// TwinCAT 3 PLC project R2_SafetyPLC
// ProgramVersion: 3.1.4022.3
// libraries:
//   Tc2_EtherCAT, * (Beckhoff Automation GmbH)
//   Tc2_Standard, * (Beckhoff Automation GmbH)
//   Tc2_System, * (Beckhoff Automation GmbH)
//   Tc2_Utilities, * (Beckhoff Automation GmbH)
//   Tc3_Module, * (Beckhoff Automation GmbH)
//   VisuDialogs, * (System)
// project tree:
//   DUTs/FBs/Enums/ E_SAFETY_FBState.TcDUT, E_SAFETY_FBStateCS.TcDUT, E_SAFETY_FBStateMUTING.TcDUT, E_SAFETY_FBStateSetReset.TcDUT, E_SAFETY_FBStateTimer.TcDUT
//   DUTs/FBs/FBStatus/ ST_Empty.TcDUT, ST_SAFETY_AND.TcDUT, ST_SAFETY_CONNECTIONSHUTDOWN.TcDUT, ST_SAFETY_DECOUPLE.TcDUT, ST_SAFETY_EDM.TcDUT, ST_SAFETY_ESTOP.TcDUT, ST_SAFETY_FBStatus.TcDUT, ST_SAFETY_MON.TcDUT, ST_SAFETY_MUTING.TcDUT, ST_SAFETY_OPMODE.TcDUT, ST_SAFETY_OR.TcDUT, ST_SAFETY_RS.TcDUT, ST_SAFETY_SR.TcDUT, ST_SAFETY_TOF.TcDUT, ST_SAFETY_TON.TcDUT, ST_SAFETY_TWOHAND.TcDUT
//   DUTs/FBs/ ST_SAFETY_FBAND.TcDUT, ST_SAFETY_FBCONNECTIONSHUTDOWN.TcDUT, ST_SAFETY_FBDECOUPLE.TcDUT, ST_SAFETY_FBEDM.TcDUT, ST_SAFETY_FBESTOP.TcDUT, ST_SAFETY_FBMON.TcDUT, ST_SAFETY_FBMUTING.TcDUT, ST_SAFETY_FBOPMODE.TcDUT, ST_SAFETY_FBOR.TcDUT, ST_SAFETY_FBRS.TcDUT, ST_SAFETY_FBSR.TcDUT, ST_SAFETY_FBTOF.TcDUT, ST_SAFETY_FBTON.TcDUT, ST_SAFETY_FBTWOHAND.TcDUT
//   DUTs/FBs/Unions/ U_SAFETY_AND.TcDUT, U_SAFETY_CONNECTIONSHUTDOWN.TcDUT, U_SAFETY_DECOUPLE.TcDUT, U_SAFETY_EDM.TcDUT, U_SAFETY_ESTOP.TcDUT, U_SAFETY_MON.TcDUT, U_SAFETY_MUTING.TcDUT, U_SAFETY_OPMODE.TcDUT, U_SAFETY_OR.TcDUT, U_SAFETY_RS.TcDUT, U_SAFETY_SR.TcDUT, U_SAFETY_TOF.TcDUT, U_SAFETY_TON.TcDUT, U_SAFETY_TWOHAND.TcDUT
//   DUTs/HW/ E_AX580x_ERROR.TcDUT, ST_AX580x_DiagnosticData.TcDUT, ST_EL1904_DiagnosticData.TcDUT, ST_EL2904_DiagnosticData.TcDUT, ST_EL6900_DiagnosticData.TcDUT, ST_EL6900_StatusData.TcDUT, ST_ELxxxx_Data.TcDUT
//   DUTs/Others/ E_SAFETY_ConnectionDiag.TcDUT, E_SAFETY_ConnectionState.TcDUT, E_SAFETY_GroupState.TcDUT, E_SAFETY_ProjectState.TcDUT, ST_SAFETYGroupIO.TcDUT, ST_SAFETYStatusConnection.TcDUT, ST_SAFETYStatusGroup.TcDUT
//   / GlobalTextList.TcGTLO, SafetyTask.TcTTO, Visualization Manager.TcVMO (not stored)
//   POUs/FBs/ F_SAFETY_StatusFB_TO_AND.TcPOU, F_SAFETY_StatusFB_TO_CONNECTIONSHUTDOWN.TcPOU, F_SAFETY_StatusFB_TO_DECOUPLE.TcPOU, F_SAFETY_StatusFB_TO_EDM.TcPOU, F_SAFETY_StatusFB_TO_ESTOP.TcPOU, F_SAFETY_StatusFB_TO_MON.TcPOU, F_SAFETY_StatusFB_TO_MUTING.TcPOU, F_SAFETY_StatusFB_TO_OPMODE.TcPOU, F_SAFETY_StatusFB_TO_OR.TcPOU, F_SAFETY_StatusFB_TO_RS.TcPOU, F_SAFETY_StatusFB_TO_SR.TcPOU, F_SAFETY_StatusFB_TO_TOF.TcPOU, F_SAFETY_StatusFB_TO_TON.TcPOU, F_SAFETY_StatusFB_TO_TWOHAND.TcPOU
//   POUs/HW/ FB_AX580x_DiagnosticData.TcPOU, FB_EL1904_DiagnosticData.TcPOU, FB_EL2904_DiagnosticData.TcPOU, FB_EL6900_DiagnosticData.TcPOU, FB_EL6900_StatusData.TcPOU
//   POUs/ MAINSafety.TcPOU
//   POUs/Others/ FB_SAFETY_AutoGroupErrACK.TcPOU, F_SAFETY_DOUBLESWAPDWORD.TcPOU, F_SAFETY_DWORD_TO_STIRNGHEX.TcPOU, I_ErrorHandling.TcIO
//   Version/ F_GetVersionSafetyDiag.TcPOU, Global_Version.TcGVL
//   VISUs/FBs/ TL_ConnectionDiag.TcTLO, TL_ConnectionState.TcTLO, TL_FbState.TcTLO, TL_FbStateCS.TcTLO, TL_FbStateMUTING.TcTLO, TL_FbStateSetReset.TcTLO, TL_FbStateTimer.TcTLO, TL_GroupState.TcTLO, V_PH_AND.TcVIS, V_PH_CONNECTIONSHUTDOWN.TcVIS, V_PH_DECOUPLE.TcVIS, V_PH_EDM.TcVIS, V_PH_ESTOP.TcVIS, V_PH_MON.TcVIS, V_PH_MUTING.TcVIS, V_PH_OPMODE.TcVIS, V_PH_OR.TcVIS, V_PH_RS.TcVIS, V_PH_SR.TcVIS, V_PH_TOF.TcVIS, V_PH_TON.TcVIS, V_PH_TWOHAND.TcVIS
//   VISUs/HW/ V_PH_EL1904_DIAG.TcVIS, V_PH_EL2904_DIAG.TcVIS, V_PH_EL6900_DIAG.TcVIS
//   VISUs/ V_PH_CONNECTION.TcVIS, V_PH_GROUP.TcVIS
// (motion and I/O tree: see PLC project r1_templateplc)
// real-time tasks:
//   TASK PlcTask: cycle T#10ms, priority 20, ADS port 350
//   TASK SafetyTask: cycle T#10ms, priority 21, ADS port 351

CONFIGURATION R2_SafetyPLC
    RESOURCE PLC ON TwinCAT3
        TASK SafetyTask(INTERVAL := T#10ms, PRIORITY := 21);
        PROGRAM MAINSafety WITH SafetyTask : MAINSafety;
    END_RESOURCE
END_CONFIGURATION

// ---- DUTs/FBs/Enums/E_SAFETY_FBState.TcDUT
TYPE E_SAFETY_FBState :
(* Refers to the following function blocks: AND, OR, OPMODE, ESTOP, MON, DECOUPLE, TWO-HAND, EDM *)
(
	eSAFETY_FBState_UNDEFINED		:= 0,
	eSAFETY_FBState_RUN				:= 1,
	eSAFETY_FBState_STOP 			:= 2,
	eSAFETY_FBState_SAFE 			:= 3,
	eSAFETY_FBState_ERROR 			:= 4,
	eSAFETY_FBState_RESET 			:= 5,
	eSAFETY_FBState_START 			:= 6,
	eSAFETY_FBState_ERRORDELAY		:= 7,
	eSAFETY_FBState_DELAYOUT		:= 8,
	eSAFETY_FBState_FUNCTEST		:= 9,
	eSAFETY_FBState_1BUTTON			:= 11,
	eSAFETY_FBState_2BUTTON			:= 12,
	eSAFETY_FBState_RELEASE			:= 13,
	eSAFETY_FBState_MONOFF			:= 14,
	eSAFETY_FBState_MONON			:= 15
);
END_TYPE

// ---- DUTs/FBs/Enums/E_SAFETY_FBStateCS.TcDUT
TYPE E_SAFETY_FBStateCS :
(* Refers to the following function blocks: CONNECTION SHUTDOWN *)
(
	eSAFETY_FBStateCS_UNDEFINED			:= 0,
	eSAFETY_FBStateCS_RUN				:= 1,
	eSAFETY_FBStateCS_STOP 				:= 2,
	eSAFETY_FBStateCS_SAFE 				:= 3,
	eSAFETY_FBStateCS_ERROR 			:= 4,
	eSAFETY_FBStateCS_RESET				:= 5,
	eSAFETY_FBStateCS_ACTIVE			:= 10,
	eSAFETY_FBStateCS_DEACTIVE			:= 11
);
END_TYPE

// ---- DUTs/FBs/Enums/E_SAFETY_FBStateMUTING.TcDUT
TYPE E_SAFETY_FBStateMUTING :
(* Refers to the following function blocks: MUTING *)
(
	eSAFETY_FBStateMUTING_UNDEFINED		:= 0,
	eSAFETY_FBStateMUTING_RUN 			:= 1,
	eSAFETY_FBStateMUTING_STOP 			:= 2,
	eSAFETY_FBStateMUTING_SAFE 			:= 3,
	eSAFETY_FBStateMUTING_ERROR 		:= 4,
	eSAFETY_FBStateMUTING_RESET			:= 5,
	eSAFETY_FBStateMUTING_DELAYOUT		:= 8,
	eSAFETY_FBStateMUTING_MUTING1		:= 9,
	eSAFETY_FBStateMUTING_MUTING2		:= 10,
	eSAFETY_FBStateMUTING_MUTING3		:= 11,
	eSAFETY_FBStateMUTING_MUTING4		:= 12,
	eSAFETY_FBStateMUTING_MUTING5		:= 13,
	eSAFETY_FBStateMUTING_MUTING6		:= 14,
	eSAFETY_FBStateMUTING_MUTING7		:= 15,
	eSAFETY_FBStateMUTING_MUTING8		:= 16,
	eSAFETY_FBStateMUTING_MUTING9		:= 17
);
END_TYPE

// ---- DUTs/FBs/Enums/E_SAFETY_FBStateSetReset.TcDUT
TYPE E_SAFETY_FBStateSetReset :
(* Refers to the following function blocks: SR, RS *)
(
	eSAFETY_FBStateSetReset_UNDEFINED 	:= 0,
	eSAFETY_FBStateSetReset_STOP 		:= 2,
	eSAFETY_FBStateSetReset_SAFE 		:= 3,
	eSAFETY_FBStateSetReset_SET 		:= 9
);
END_TYPE

// ---- DUTs/FBs/Enums/E_SAFETY_FBStateTimer.TcDUT
TYPE E_SAFETY_FBStateTimer :
(* Refers to the following function blocks: TON, TOF *)
(
	eSAFETY_FBStateTimer_UNDEFINED 	:= 0,
	eSAFETY_FBStateTimer_RUN 		:= 1,
	eSAFETY_FBStateTimer_STOP 		:= 2,
	eSAFETY_FBStateTimer_SAFE 		:= 3,
	eSAFETY_FBStateTimer_DELAYOUT 	:= 8,
	eSAFETY_FBStateTimer_DELAYIN 	:= 9
);
END_TYPE

// ---- DUTs/FBs/FBStatus/ST_Empty.TcDUT
TYPE ST_Empty :
STRUCT
	{attribute 'hide'}
	BUnknown						: BYTE;
	BState							: BYTE;
(* wDiagnosis *)
	{attribute 'hide'}
	bDiagBIT0						: BIT; 		(* Empty *)
	{attribute 'hide'}
	bDiagBIT1						: BIT; 		(* Empty *)
	{attribute 'hide'}
	bDiagBIT2						: BIT; 		(* Empty *)
	{attribute 'hide'}
	bDiagBIT3						: BIT; 		(* Empty *)
	{attribute 'hide'}
	bDiagBIT4						: BIT; 		(* Empty *)
	{attribute 'hide'}
	bDiagBIT5						: BIT; 		(* Empty *)
	{attribute 'hide'}
	bDiagBIT6						: BIT; 		(* Empty *)
	{attribute 'hide'}
	bDiagBIT7						: BIT; 		(* Empty *)
	{attribute 'hide'}
	bDiagBIT8						: BIT; 		(* Empty *)
	{attribute 'hide'}
	bDiagBIT9						: BIT; 		(* Empty *)
	{attribute 'hide'}
	bDiagBIT10						: BIT; 		(* Empty *)
	{attribute 'hide'}
	bDiagBIT11						: BIT; 		(* Empty *)
	{attribute 'hide'}
	bDiagBIT12						: BIT; 		(* Empty *)
	{attribute 'hide'}
	bDiagBIT13						: BIT; 		(* Empty *)
	{attribute 'hide'}
	bDiagBIT14						: BIT; 		(* Empty *)
	{attribute 'hide'}
	bDiagBIT15						: BIT; 		(* Empty *)
(* wInputs *)
	{attribute 'hide'}
	bInputBIT0						: BIT; 		(* Empty *)
	{attribute 'hide'}
	bInputBIT1						: BIT; 		(* Empty *)
	{attribute 'hide'}
	bInputBIT2						: BIT; 		(* Empty *)
	{attribute 'hide'}
	bInputBIT3						: BIT; 		(* Empty *)
	{attribute 'hide'}
	bInputBIT4						: BIT; 		(* Empty *)
	{attribute 'hide'}
	bInputBIT5						: BIT; 		(* Empty *)
	{attribute 'hide'}
	bInputBIT6						: BIT; 		(* Empty *)
	{attribute 'hide'}
	bInputBIT7						: BIT; 		(* Empty *)
	{attribute 'hide'}
	bInputBIT8						: BIT; 		(* Empty *)
	{attribute 'hide'}
	bInputBIT9						: BIT; 		(* Empty *)
	{attribute 'hide'}
	bInputBIT10						: BIT; 		(* Empty *)
	{attribute 'hide'}
	bInputBIT11						: BIT; 		(* Empty *)
	{attribute 'hide'}
	bInputBIT12						: BIT; 		(* Empty *)
	{attribute 'hide'}
	bInputBIT13						: BIT; 		(* Empty *)
	{attribute 'hide'}
	bInputBIT14						: BIT; 		(* Empty *)
	{attribute 'hide'}
	bInputBIT15						: BIT; 		(* Empty *)
(* wOutputs *)
	{attribute 'hide'}
	bOutputBIT0						: BIT; 		(* Empty *)
	{attribute 'hide'}
	bOutputBIT1						: BIT; 		(* Empty *)
	{attribute 'hide'}
	bOutputBIT2						: BIT; 		(* Empty *)
	{attribute 'hide'}
	bOutputBIT3						: BIT; 		(* Empty *)
	{attribute 'hide'}
	bOutputBIT4						: BIT; 		(* Empty *)
	{attribute 'hide'}
	bOutputBIT5						: BIT; 		(* Empty *)
	{attribute 'hide'}
	bOutputBIT6						: BIT; 		(* Empty *)
	{attribute 'hide'}
	bOutputBIT7						: BIT; 		(* Empty *)
	{attribute 'hide'}
	bOutputBIT8						: BIT; 		(* Empty *)
	{attribute 'hide'}
	bOutputBIT9						: BIT; 		(* Empty *)
	{attribute 'hide'}
	bOutputBIT10					: BIT; 		(* Empty *)
	{attribute 'hide'}
	bOutputBIT11					: BIT; 		(* Empty *)
	{attribute 'hide'}
	bOutputBIT12					: BIT; 		(* Empty *)
	{attribute 'hide'}
	bOutputBIT13					: BIT; 		(* Empty *)
	{attribute 'hide'}
	bOutputBIT14					: BIT; 		(* Empty *)
	{attribute 'hide'}
	bOutputBIT15					: BIT; 		(* Empty *)
END_STRUCT
END_TYPE

// ---- DUTs/FBs/FBStatus/ST_SAFETY_AND.TcDUT
//UPDATE: Zamiana dwóch pierwszych bitów zmiennej wOutputs
TYPE ST_SAFETY_AND :
STRUCT
	{attribute 'hide'}
	BUnknown						: BYTE;
	BState							: BYTE;
(* wDiagnosis *)
	{attribute 'hide'}
	bDiagBIT0						: BIT; 		(* Empty *)
	{attribute 'hide'}
	bDiagBIT1						: BIT; 		(* Empty *)
	{attribute 'hide'}
	bDiagBIT2						: BIT; 		(* Empty *)
	{attribute 'hide'}
	bDiagBIT3						: BIT; 		(* Empty *)
	{attribute 'hide'}
	bDiagBIT4						: BIT; 		(* Empty *)
	{attribute 'hide'}
	bDiagBIT5						: BIT; 		(* Empty *)
	{attribute 'hide'}
	bDiagBIT6						: BIT; 		(* Empty *)
	{attribute 'hide'}
	bDiagBIT7						: BIT; 		(* Empty *)
	{attribute 'hide'}
	bDiagBIT8						: BIT; 		(* Empty *)
	{attribute 'hide'}
	bDiagBIT9						: BIT; 		(* Empty *)
	{attribute 'hide'}
	bDiagBIT10						: BIT; 		(* Empty *)
	{attribute 'hide'}
	bDiagBIT11						: BIT; 		(* Empty *)
	{attribute 'hide'}
	bDiagBIT12						: BIT; 		(* Empty *)
	{attribute 'hide'}
	bDiagBIT13						: BIT; 		(* Empty *)
	{attribute 'hide'}
	bDiagBIT14						: BIT; 		(* Empty *)
	{attribute 'hide'}
	bDiagBIT15						: BIT; 		(* Empty *)
(* wInputs *)
	{attribute 'hide'}
	bInputBIT0						: BIT; 		(* Empty *)
	{attribute 'hide'}
	bInputBIT1						: BIT; 		(* Empty *)
	{attribute 'hide'}
	bInputBIT2						: BIT; 		(* Empty *)
	{attribute 'hide'}
	bInputBIT3						: BIT; 		(* Empty *)
	{attribute 'hide'}
	bInputBIT4						: BIT; 		(* Empty *)
	{attribute 'hide'}
	bInputBIT5						: BIT; 		(* Empty *)
	{attribute 'hide'}
	bInputBIT6						: BIT; 		(* Empty *)
	{attribute 'hide'}
	bInputBIT7						: BIT; 		(* Empty *)
	bIn_ANDIn1						: BIT; 		(* .8 *)
	bIn_ANDIn2						: BIT; 		(* .9 *)
	bIn_ANDIn3						: BIT; 		(* .10 *)
	bIn_ANDIn4						: BIT; 		(* .11 *)
	bIn_ANDIn5						: BIT; 		(* .12 *)
	bIn_ANDIn6						: BIT; 		(* .13 *)
	bIn_ANDIn7						: BIT; 		(* .14 *)
	bIn_ANDIn8						: BIT; 		(* .15 *)
(* wOutputs *)
	{attribute 'hide'}
	bOut_ANDOut_OLD					: BIT; 		(* .0 UPDATE: Empty*)
	//{attribute 'hide'}
	bOut_ANDOut						: BIT; 		(* .1 UPDATE: AND_OUT*)
	{attribute 'hide'}
	bOutputBIT2						: BIT; 		(* Empty *)
	{attribute 'hide'}
	bOutputBIT3						: BIT; 		(* Empty *)
	{attribute 'hide'}
	bOutputBIT4						: BIT; 		(* Empty *)
	{attribute 'hide'}
	bOutputBIT5						: BIT; 		(* Empty *)
	{attribute 'hide'}
	bOutputBIT6						: BIT; 		(* Empty *)
	{attribute 'hide'}
	bOutputBIT7						: BIT; 		(* Empty *)
	{attribute 'hide'}
	bOutputBIT8						: BIT; 		(* Empty *)
	{attribute 'hide'}
	bOutputBIT9						: BIT; 		(* Empty *)
	{attribute 'hide'}
	bOutputBIT10					: BIT; 		(* Empty *)
	{attribute 'hide'}
	bOutputBIT11					: BIT; 		(* Empty *)
	{attribute 'hide'}
	bOutputBIT12					: BIT; 		(* Empty *)
	{attribute 'hide'}
	bOutputBIT13					: BIT; 		(* Empty *)
	{attribute 'hide'}
	bOutputBIT14					: BIT; 		(* Empty *)
	{attribute 'hide'}
	bOutputBIT15					: BIT; 		(* Empty *)
END_STRUCT
END_TYPE

// ---- DUTs/FBs/FBStatus/ST_SAFETY_CONNECTIONSHUTDOWN.TcDUT
TYPE ST_SAFETY_CONNECTIONSHUTDOWN :
STRUCT
	{attribute 'hide'}
	BUnknown						: BYTE;
	BState							: BYTE;
(* wDiagnosis *)
	
	bDiag_DiscErrorCS1_2			: BIT;  	(* Discrepancy error input group 1 *)
	{attribute 'hide'}
	bDiagBIT1						: BIT; 		(* Empty *)
	{attribute 'hide'}
	bDiagBIT2						: BIT; 		(* Empty *)
	{attribute 'hide'}
	bDiagBIT3						: BIT; 		(* Empty *)
	{attribute 'hide'}
	bDiagBIT4						: BIT; 		(* Empty *)
	{attribute 'hide'}
	bDiagBIT5						: BIT; 		(* Empty *)
	{attribute 'hide'}
	bDiagBIT6						: BIT; 		(* Empty *)
	{attribute 'hide'}
	bDiagBIT7						: BIT; 		(* Empty *)
	{attribute 'hide'}
	bDiagBIT8						: BIT; 		(* Empty *)
	{attribute 'hide'}
	bDiagBIT9						: BIT; 		(* Empty *)
	{attribute 'hide'}
	bDiagBIT10						: BIT; 		(* Empty *)
	{attribute 'hide'}
	bDiagBIT11						: BIT; 		(* Empty *)
	{attribute 'hide'}
	bDiagBIT12						: BIT; 		(* Empty *)
	{attribute 'hide'}
	bDiagBIT13						: BIT; 		(* Empty *)
	{attribute 'hide'}
	bDiagBIT14						: BIT; 		(* Empty *)
	{attribute 'hide'}
	bDiagBIT15						: BIT; 		(* Empty *)
(* wInputs *)
	{attribute 'hide'}
	bInputBIT0						: BIT; 		(* Empty *)
	{attribute 'hide'}
	bInputBIT1						: BIT; 		(* Empty *)
	{attribute 'hide'}
	bInputBIT2						: BIT; 		(* Empty *)
	{attribute 'hide'}
	bInputBIT3						: BIT; 		(* Empty *)
	{attribute 'hide'}
	bInputBIT4						: BIT; 		(* Empty *)
	{attribute 'hide'}
	bInputBIT5						: BIT; 		(* Empty *)
	{attribute 'hide'}
	bInputBIT6						: BIT; 		(* Empty *)
	{attribute 'hide'}
	bInputBIT7						: BIT; 		(* Empty *)
	bIn_Deactivate1					: BIT; 		(* .8 *)
	bIn_Deactivate2					: BIT; 		(* .9 *)
	{attribute 'hide'}
	bInputBIT10						: BIT; 		(* Empty *)
	{attribute 'hide'}
	bInputBIT11						: BIT; 		(* Empty *)
	{attribute 'hide'}
	bInputBIT12						: BIT; 		(* Empty *)
	{attribute 'hide'}
	bInputBIT13						: BIT; 		(* Empty *)
	{attribute 'hide'}
	bInputBIT14						: BIT; 		(* Empty *)
	{attribute 'hide'}
	bInputBIT15						: BIT; 		(* Empty *)
(* wOutputs *)
	bOut_Error						: BOOL; 	(* .0 *)
	bOut_Deactivated				: BOOL; 	(* .1 *)
	{attribute 'hide'}
	bOutputBIT2						: BIT; 		(* Empty *)
	{attribute 'hide'}
	bOutputBIT3						: BIT; 		(* Empty *)
	{attribute 'hide'}
	bOutputBIT4						: BIT; 		(* Empty *)
	{attribute 'hide'}
	bOutputBIT5						: BIT; 		(* Empty *)
	{attribute 'hide'}
	bOutputBIT6						: BIT; 		(* Empty *)
	{attribute 'hide'}
	bOutputBIT7						: BIT; 		(* Empty *)
	{attribute 'hide'}
	bOutputBIT8						: BIT; 		(* Empty *)
	{attribute 'hide'}
	bOutputBIT9						: BIT; 		(* Empty *)
	{attribute 'hide'}
	bOutputBIT10					: BIT; 		(* Empty *)
	{attribute 'hide'}
	bOutputBIT11					: BIT; 		(* Empty *)
	{attribute 'hide'}
	bOutputBIT12					: BIT; 		(* Empty *)
	{attribute 'hide'}
	bOutputBIT13					: BIT; 		(* Empty *)
	{attribute 'hide'}
	bOutputBIT14					: BIT; 		(* Empty *)
	{attribute 'hide'}
	bOutputBIT15					: BIT; 		(* Empty *)
END_STRUCT
END_TYPE

// ---- DUTs/FBs/FBStatus/ST_SAFETY_DECOUPLE.TcDUT
TYPE ST_SAFETY_DECOUPLE :
STRUCT
	{attribute 'hide'}
	BUnknown						: BYTE;
	BState							: BYTE;
(* wDiagnosis *)
	{attribute 'hide'}
	bDiagBIT0						: BIT; 		(* Empty *)
	{attribute 'hide'}
	bDiagBIT1						: BIT; 		(* Empty *)
	{attribute 'hide'}
	bDiagBIT2						: BIT; 		(* Empty *)
	{attribute 'hide'}
	bDiagBIT3						: BIT; 		(* Empty *)
	{attribute 'hide'}
	bDiagBIT4						: BIT; 		(* Empty *)
	{attribute 'hide'}
	bDiagBIT5						: BIT; 		(* Empty *)
	{attribute 'hide'}
	bDiagBIT6						: BIT; 		(* Empty *)
	{attribute 'hide'}
	bDiagBIT7						: BIT; 		(* Empty *)
	{attribute 'hide'}
	bDiagBIT8						: BIT; 		(* Empty *)
	{attribute 'hide'}
	bDiagBIT9						: BIT; 		(* Empty *)
	{attribute 'hide'}
	bDiagBIT10						: BIT; 		(* Empty *)
	{attribute 'hide'}
	bDiagBIT11						: BIT; 		(* Empty *)
	{attribute 'hide'}
	bDiagBIT12						: BIT; 		(* Empty *)
	{attribute 'hide'}
	bDiagBIT13						: BIT; 		(* Empty *)
	{attribute 'hide'}
	bDiagBIT14						: BIT; 		(* Empty *)
	{attribute 'hide'}
	bDiagBIT15						: BIT; 		(* Empty *)
(* wInputs *)
	{attribute 'hide'}
	bInputBIT0						: BIT; 		(* Empty *)
	{attribute 'hide'}
	bInputBIT1						: BIT; 		(* Empty *)
	{attribute 'hide'}
	bInputBIT2						: BIT; 		(* Empty *)
	{attribute 'hide'}
	bInputBIT3						: BIT; 		(* Empty *)
	{attribute 'hide'}
	bInputBIT4						: BIT; 		(* Empty *)
	{attribute 'hide'}
	bInputBIT5						: BIT; 		(* Empty *)
	{attribute 'hide'}
	bInputBIT6						: BIT; 		(* Empty *)
	{attribute 'hide'}
	bInputBIT7						: BIT; 		(* Empty *)
	bIn_DECOUPLEIn1					: BIT; 		(* .8 *)
	bIn_DECOUPLEIn2					: BIT; 		(* .9 *)
	bIn_DECOUPLEIn3					: BIT; 		(* .10 *)
	bIn_DECOUPLEIn4					: BIT; 		(* .11 *)
	bIn_DECOUPLEIn5					: BIT; 		(* .12 *)
	bIn_DECOUPLEIn6					: BIT; 		(* .13 *)
	bIn_DECOUPLEIn7					: BIT; 		(* .14 *)
	bIn_DECOUPLEIn8					: BIT; 		(* .15 *)
(* wOutputs *)
	{attribute 'hide'}
	bOutputBIT0						: BIT; 		(* Empty *)
	{attribute 'hide'}
	bOutputBIT1						: BIT; 		(* Empty *)
	{attribute 'hide'}
	bOutputBIT2						: BIT; 		(* Empty *)
	{attribute 'hide'}
	bOutputBIT3						: BIT; 		(* Empty *)
	{attribute 'hide'}
	bOutputBIT4						: BIT; 		(* Empty *)
	{attribute 'hide'}
	bOutputBIT5						: BIT; 		(* Empty *)
	{attribute 'hide'}
	bOutputBIT6						: BIT; 		(* Empty *)
	{attribute 'hide'}
	bOutputBIT7						: BIT; 		(* Empty *)
	bOut_DECOUPLEOut1				: BOOL; 	(* .8 *)
	bOut_DECOUPLEOut2				: BOOL; 	(* .9 *)
	bOut_DECOUPLEOut3				: BOOL; 	(* .10 *)
	bOut_DECOUPLEOut4				: BOOL; 	(* .11 *)
	bOut_DECOUPLEOut5				: BOOL; 	(* .12 *)
	bOut_DECOUPLEOut6				: BOOL; 	(* .13 *)
	bOut_DECOUPLEOut7				: BOOL; 	(* .14 *)
	bOut_DECOUPLEOut8				: BOOL; 	(* .15 *)
END_STRUCT
END_TYPE

// ---- DUTs/FBs/FBStatus/ST_SAFETY_EDM.TcDUT
TYPE ST_SAFETY_EDM :
STRUCT
	{attribute 'hide'}
	BUnknown						: BYTE;
	BState							: BYTE;
(* wDiagnosis *)
	bDiag_SwitchOffError			: BIT; 		(* Switch-OFF timer elapsed  *)
	bDiag_SwitchOnError				: BIT; 		(* Switch-ON timer elapsed  *)
	{attribute 'hide'}
	bDiagBIT2						: BIT; 		(* Empty *)
	{attribute 'hide'}
	bDiagBIT3						: BIT; 		(* Empty *)
	{attribute 'hide'}
	bDiagBIT4						: BIT; 		(* Empty *)
	{attribute 'hide'}
	bDiagBIT5						: BIT; 		(* Empty *)
	{attribute 'hide'}
	bDiagBIT6						: BIT; 		(* Empty *)
	{attribute 'hide'}
	bDiagBIT7						: BIT; 		(* Empty *)
	{attribute 'hide'}
	bDiagBIT8						: BIT; 		(* Empty *)
	{attribute 'hide'}
	bDiagBIT9						: BIT; 		(* Empty *)
	{attribute 'hide'}
	bDiagBIT10						: BIT; 		(* Empty *)
	{attribute 'hide'}
	bDiagBIT11						: BIT; 		(* Empty *)
	{attribute 'hide'}
	bDiagBIT12						: BIT; 		(* Empty *)
	{attribute 'hide'}
	bDiagBIT13						: BIT; 		(* Empty *)
	{attribute 'hide'}
	bDiagBIT14						: BIT; 		(* Empty *)
	{attribute 'hide'}
	bDiagBIT15						: BIT; 		(* Empty *)
(* wInputs *)
	{attribute 'hide'}
	bInputBIT0						: BIT; 		(* Empty *)
	{attribute 'hide'}
	bInputBIT1						: BIT; 		(* Empty *)
	{attribute 'hide'}
	bInputBIT2						: BIT; 		(* Empty *)
	{attribute 'hide'}
	bInputBIT3						: BIT; 		(* Empty *)
	{attribute 'hide'}
	bInputBIT4						: BIT; 		(* Empty *)
	{attribute 'hide'}
	bInputBIT5						: BIT; 		(* Empty *)
	{attribute 'hide'}
	bInputBIT6						: BIT; 		(* Empty *)
	{attribute 'hide'}
	bInputBIT7						: BIT; 		(* Empty *)
	bIn_MON1						: BIT; 		(* .8 *)
	bIn_MON2						: BIT; 		(* .9 *)
	{attribute 'hide'}
	bInputBIT10						: BIT; 		(* Empty *)
	{attribute 'hide'}
	bInputBIT11						: BIT; 		(* Empty *)
	{attribute 'hide'}
	bInputBIT12						: BIT; 		(* Empty *)
	{attribute 'hide'}
	bInputBIT13						: BIT; 		(* Empty *)
	{attribute 'hide'}
	bInputBIT14						: BIT; 		(* Empty *)
	{attribute 'hide'}
	bInputBIT15						: BIT; 		(* Empty *)
(* wOutputs *)
	bOut_Error						: BIT; 		(* .0 *)
	{attribute 'hide'}
	bOutputBIT1						: BIT; 		(* Empty *)
	{attribute 'hide'}
	bOutputBIT2						: BIT; 		(* Empty *)
	{attribute 'hide'}
	bOutputBIT3						: BIT; 		(* Empty *)
	{attribute 'hide'}
	bOutputBIT4						: BIT; 		(* Empty *)
	{attribute 'hide'}
	bOutputBIT5						: BIT; 		(* Empty *)
	{attribute 'hide'}
	bOutputBIT6						: BIT; 		(* Empty *)
	{attribute 'hide'}
	bOutputBIT7						: BIT; 		(* Empty *)
	{attribute 'hide'}
	bOutputBIT8						: BIT; 		(* Empty *)
	{attribute 'hide'}
	bOutputBIT9						: BIT; 		(* Empty *)
	{attribute 'hide'}
	bOutputBIT10					: BIT; 		(* Empty *)
	{attribute 'hide'}
	bOutputBIT11					: BIT; 		(* Empty *)
	{attribute 'hide'}
	bOutputBIT12					: BIT; 		(* Empty *)
	{attribute 'hide'}
	bOutputBIT13					: BIT; 		(* Empty *)
	{attribute 'hide'}
	bOutputBIT14					: BIT; 		(* Empty *)
	{attribute 'hide'}
	bOutputBIT15					: BIT; 		(* Empty *)
END_STRUCT
END_TYPE

// ---- DUTs/FBs/FBStatus/ST_SAFETY_ESTOP.TcDUT
TYPE ST_SAFETY_ESTOP :
STRUCT
	{attribute 'hide'}
	BUnknown						: BYTE;
	BState							: BYTE;
(* wDiagnosis *)
	bDiag_DiscError1_2				: BIT;		(* Bit 0: Discrepancy error input group 1 (EStopIn1/2) *)
	bDiag_DiscError3_4				: BIT;		(* Bit 1: Discrepancy error input group 2 (EStopIn3/4) *)
	bDiag_DiscError5_6				: BIT;		(* Bit 2: Discrepancy error input group 2 (EStopIn5/6) *)
	bDiag_DiscError7_8				: BIT;		(* Bit 3: Discrepancy error input group 2 (EStopIn7/8) *)
	bDiag_EDM1Error					: BIT;		(* Bit 4: EDM monitoring error EDM1 Error *)
	bDiag_EDM2Error					: BIT;		(* Bit 5: EDM monitoring error EDM2 Error *)
	{attribute 'hide'}
	bDiagBIT6						: BIT; 		(* Empty *)
	{attribute 'hide'}
	bDiagBIT7						: BIT; 		(* Empty *)
	bDiag_DiscErrorSIADE1_2			: BIT;		(* Bit 8: Discrepancy error input group 1 with activated option "Safe Inputs after Disc Error"  (set in addition to bit 0) *)
	bDiag_DiscErrorSIADE3_4			: BIT;		(* Bit 9: Discrepancy error input group 2 with activated option "Safe Inputs after Disc Error"  (set in addition to bit 1) *)
	bDiag_DiscErrorSIADE5_6			: BIT;		(* Bit 10: Discrepancy error input group 3 with activated option "Safe Inputs after Disc Error"  (set in addition to bit 2) *)
	bDiag_DiscErrorSIADE7_8			: BIT;		(* Bit 11: Discrepancy error input group 4 with activated option "Safe Inputs after Disc Error"  (set in addition to bit 3)*)
	{attribute 'hide'}
	bDiagBIT12						: BIT; 		(* Empty *)
	{attribute 'hide'}
	bDiagBIT13						: BIT; 		(* Empty *)
	{attribute 'hide'}
	bDiagBIT14						: BIT; 		(* Empty *)
	{attribute 'hide'}
	bDiagBIT15						: BIT; 		(* Empty *)
(* wInputs *)
	bIn_Restart						: BIT; 		(* .0 *)
	bIn_EDM1						: BIT; 		(* .1 *)
	bIn_EDM2						: BIT; 		(* .2 *)
	{attribute 'hide'}
	bInputBIT3						: BIT; 		(* Empty *)
	{attribute 'hide'}
	bInputBIT4						: BIT; 		(* Empty *)
	{attribute 'hide'}
	bInputBIT5						: BIT; 		(* Empty *)
	{attribute 'hide'}
	bInputBIT6						: BIT; 		(* Empty *)
	{attribute 'hide'}
	bInputBIT7						: BIT; 		(* Empty *)
	bIn_EStopIn1					: BIT; 		(* .8 *)
	bIn_EStopIn2					: BIT; 		(* .9 *)
	bIn_EStopIn3					: BIT; 		(* .10 *)
	bIn_EStopIn4					: BIT; 		(* .11 *)
	bIn_EStopIn5					: BIT; 		(* .12 *)
	bIn_EStopIn6					: BIT; 		(* .13 *)
	bIn_EStopIn7					: BIT; 		(* .14 *)
	bIn_EStopIn8					: BIT; 		(* .15 *)
(* wOutputs *)
	bOut_Error						: BIT; 		(* .0 *)
	bOut_EstopOut					: BIT; 		(* .1 *)
	bOut_EstopDelOut				: BIT; 		(* .2 *)
	{attribute 'hide'}
	bOutputBIT3						: BIT; 		(* Empty *)
	{attribute 'hide'}
	bOutputBIT4						: BIT; 		(* Empty *)
	{attribute 'hide'}
	bOutputBIT5						: BIT; 		(* Empty *)
	{attribute 'hide'}
	bOutputBIT6						: BIT; 		(* Empty *)
	{attribute 'hide'}
	bOutputBIT7						: BIT; 		(* Empty *)
	{attribute 'hide'}
	bOutputBIT8						: BIT; 		(* Empty *)
	{attribute 'hide'}
	bOutputBIT9						: BIT; 		(* Empty *)
	{attribute 'hide'}
	bOutputBIT10					: BIT; 		(* Empty *)
	{attribute 'hide'}
	bOutputBIT11					: BIT; 		(* Empty *)
	{attribute 'hide'}
	bOutputBIT12					: BIT; 		(* Empty *)
	{attribute 'hide'}
	bOutputBIT13					: BIT; 		(* Empty *)
	{attribute 'hide'}
	bOutputBIT14					: BIT; 		(* Empty *)
	{attribute 'hide'}
	bOutputBIT15					: BIT; 		(* Empty *)
END_STRUCT
END_TYPE

// ---- DUTs/FBs/FBStatus/ST_SAFETY_FBStatus.TcDUT
TYPE ST_SAFETY_FBStatus :
STRUCT
	BUnknown						: BYTE;
	BState							: BYTE;
	wDiagnosis						: WORD;
	wInputs							: WORD; (* 1B - Restart, EDM... 2B - Safe inputs *)
	wOutputs						: WORD; (* 1B - Error, EDM... 2B - Safe inputs  *)
END_STRUCT
END_TYPE

// ---- DUTs/FBs/FBStatus/ST_SAFETY_MON.TcDUT
TYPE ST_SAFETY_MON :
STRUCT
	{attribute 'hide'}
	BUnknown						: BYTE;
	BState							: BYTE;
(* wDiagnosis *)
	bDiag_DiscErrorMONIn1_2			: BIT; 		(* Discrepancy error input group 1 (MONIn1/2) *)
	bDiag_DiscErrorMONIn3_4			: BIT;		(* Discrepancy error input group 2 (MONIn3/4) *)
	bDiag_DiscErrorMONInSec			: BIT;		(* Discrepancy error in Secure input group (MONInSec)*) 
	{attribute 'hide'}
	bDiagBIT3						: BIT; 		(* Empty *)
	bDiag_EDM1Error					: BIT;		(* EDM monitoring error EDM1*)
	bDiag_EDM2Error					: BIT;		(* EDM monitoring error EDM2*) 
	{attribute 'hide'}
	bDiagBIT6						: BIT; 		(* Empty *)
	{attribute 'hide'}
	bDiagBIT7						: BIT; 		(* Empty *)
	{attribute 'hide'}
	bDiagBIT8						: BIT; 		(* Empty *)
	{attribute 'hide'}
	bDiagBIT9						: BIT; 		(* Empty *)
	{attribute 'hide'}
	bDiagBIT10						: BIT; 		(* Empty *)
	{attribute 'hide'}
	bDiagBIT11						: BIT; 		(* Empty *)
	{attribute 'hide'}
	bDiagBIT12						: BIT; 		(* Empty *)
	{attribute 'hide'}
	bDiagBIT13						: BIT; 		(* Empty *)
	{attribute 'hide'}
	bDiagBIT14						: BIT; 		(* Empty *)
	{attribute 'hide'}
	bDiagBIT15						: BIT; 		(* Empty *)
(* wInputs *)
	bIn_Restart						: BIT; 		(* .0 *)
	bIn_EDM1						: BIT; 		(* .1 *)
	bIn_EDM2						: BIT; 		(* .2 *)
	bIn_MONSec1						: BIT; 		(* .3 *)
	bIn_MONSec2						: BIT; 		(* .4 *)
	{attribute 'hide'}
	bInputBIT5						: BIT; 		(* Empty *)
	{attribute 'hide'}
	bInputBIT6						: BIT; 		(* Empty *)
	{attribute 'hide'}
	bInputBIT7						: BIT; 		(* Empty *)
	bIn_MONIn1						: BIT; 		(* .8 *)
	bIn_MONIn2						: BIT; 		(* .9 *)
	bIn_MONIn3						: BIT; 		(* .10 *)
	bIn_MONIn4						: BIT; 		(* .11 *)
	{attribute 'hide'}
	bInputBIT12						: BIT; 		(* Empty *)
	{attribute 'hide'}
	bInputBIT13						: BIT; 		(* Empty *)
	{attribute 'hide'}
	bInputBIT14						: BIT; 		(* Empty *)
	{attribute 'hide'}
	bInputBIT15						: BIT; 		(* Empty *)
(* wOutputs *)
	bOut_Error						: BIT; 		(* .0 *)
	bOut_MONOut						: BIT; 		(* .1 *)
	bOut_MONDelOut					: BIT; 		(* .2 *)
	{attribute 'hide'}
	bOutputBIT3						: BIT; 		(* Empty *)
	{attribute 'hide'}
	bOutputBIT4						: BIT; 		(* Empty *)
	{attribute 'hide'}
	bOutputBIT5						: BIT; 		(* Empty *)
	{attribute 'hide'}
	bOutputBIT6						: BIT; 		(* Empty *)
	{attribute 'hide'}
	bOutputBIT7						: BIT; 		(* Empty *)
	{attribute 'hide'}
	bOutputBIT8						: BIT; 		(* Empty *)
	{attribute 'hide'}
	bOutputBIT9						: BIT; 		(* Empty *)
	{attribute 'hide'}
	bOutputBIT10					: BIT; 		(* Empty *)
	{attribute 'hide'}
	bOutputBIT11					: BIT; 		(* Empty *)
	{attribute 'hide'}
	bOutputBIT12					: BIT; 		(* Empty *)
	{attribute 'hide'}
	bOutputBIT13					: BIT; 		(* Empty *)
	{attribute 'hide'}
	bOutputBIT14					: BIT; 		(* Empty *)
	{attribute 'hide'}
	bOutputBIT15					: BIT; 		(* Empty *)
END_STRUCT
END_TYPE

// ---- DUTs/FBs/FBStatus/ST_SAFETY_MUTING.TcDUT
TYPE ST_SAFETY_MUTING :
STRUCT
	{attribute 'hide'}
	BUnknown						: BYTE;
	BState							: BYTE;
(* wDiagnosis *)
	bDiag_DiscErrorMUTINGIn1_2		: BIT;		(*	Discrepancy error in muting input group 1 *)
	bDiag_DiscErrorMUTINGInOSSD		: BIT;		(*	Discrepancy error in the OSSD input group *)
	bDiag_DiscErrorMUTINGIn3_4		: BIT;		(*	Discrepancy error in muting input group 2 *)
	{attribute 'hide'}
	bDiagBIT3						: BIT; 		(* Empty *)
	bDiag_EDM1Error					: BIT;		(*	Bit 4: EDM monitoring error EDM1 Error *)
	bDiag_EDM2Error					: BIT;		(*	Bit 5: EDM monitoring error EDM2 Error *)
	bDiag_MutingSeqViolated			: BIT;		(*	Bit 6: Muting sequence was violated *)
	bDiag_MutingTimeExceeded		: BIT;		(*	Bit 7: Maximum muting time was exceeded *)
	{attribute 'hide'}
	bDiagBIT8						: BIT; 		(* Empty *)
	{attribute 'hide'}
	bDiagBIT9						: BIT; 		(* Empty *)
	{attribute 'hide'}
	bDiagBIT10						: BIT; 		(* Empty *)
	{attribute 'hide'}
	bDiagBIT11						: BIT; 		(* Empty *)
	{attribute 'hide'}
	bDiagBIT12						: BIT; 		(* Empty *)
	{attribute 'hide'}
	bDiagBIT13						: BIT; 		(* Empty *)
	{attribute 'hide'}
	bDiagBIT14						: BIT; 		(* Empty *)
	{attribute 'hide'}
	bDiagBIT15						: BIT; 		(* Empty *)
(* wInputs *)
	bIn_Enable						: BIT; 		(* .0 *)
	bIn_EDM1						: BIT; 		(* .1 *)
	bIn_EDM2						: BIT; 		(* .2 *)
	{attribute 'hide'}
	bInputBIT3						: BIT; 		(* Empty *)
	{attribute 'hide'}
	bInputBIT4						: BIT; 		(* Empty *)
	{attribute 'hide'}
	bInputBIT5						: BIT; 		(* Empty *)
	{attribute 'hide'}
	bInputBIT6						: BIT; 		(* Empty *)
	{attribute 'hide'}
	bInputBIT7						: BIT; 		(* Empty *)
	bIn_MUTINGIn1					: BIT; 		(* .8 *)
	bIn_MUTINGIn2					: BIT; 		(* .9 *)
	bIn_MUTINGIn3					: BIT; 		(* .10 *)
	bIn_MUTINGIn4					: BIT; 		(* .11 *)
	bIn_OSSDIn1						: BIT; 		(* .12 *)
	bIn_OSSDIn2						: BIT; 		(* .13 *)
	{attribute 'hide'}
	bInputBIT14						: BIT; 		(* Empty *)
	{attribute 'hide'}
	bInputBIT15						: BIT; 		(* Empty *)
(* wOutputs *)
	bOut_Error						: BIT; 		(* .0 *)
	bOut_MUTINGActive				: BIT; 		(* .1 *)
	bOut_MUTINGOut					: BIT; 		(* .2 *)
	bOut_MUTINGDelOut				: BIT; 		(* .3 *)
	{attribute 'hide'}
	bOutputBIT4						: BIT; 		(* Empty *)
	{attribute 'hide'}
	bOutputBIT5						: BIT; 		(* Empty *)
	{attribute 'hide'}
	bOutputBIT6						: BIT; 		(* Empty *)
	{attribute 'hide'}
	bOutputBIT7						: BIT; 		(* Empty *)
	{attribute 'hide'}
	bOutputBIT8						: BIT; 		(* Empty *)
	{attribute 'hide'}
	bOutputBIT9						: BIT; 		(* Empty *)
	{attribute 'hide'}
	bOutputBIT10					: BIT; 		(* Empty *)
	{attribute 'hide'}
	bOutputBIT11					: BIT; 		(* Empty *)
	{attribute 'hide'}
	bOutputBIT12					: BIT; 		(* Empty *)
	{attribute 'hide'}
	bOutputBIT13					: BIT; 		(* Empty *)
	{attribute 'hide'}
	bOutputBIT14					: BIT; 		(* Empty *)
	{attribute 'hide'}
	bOutputBIT15					: BIT; 		(* Empty *)
END_STRUCT
END_TYPE

// ---- DUTs/FBs/FBStatus/ST_SAFETY_OPMODE.TcDUT
TYPE ST_SAFETY_OPMODE :
STRUCT
	{attribute 'hide'}
	BUnknown						: BYTE;
	BState							: BYTE;
(* wDiagnosis *)
	bDiag_DiscError					: BIT; 		(* Discrepancy monitoring error *)
	{attribute 'hide'}
	bDiagBIT1						: BIT; 		(* Empty *)
	{attribute 'hide'}
	bDiagBIT2						: BIT; 		(* Empty *)
	{attribute 'hide'}
	bDiagBIT3						: BIT; 		(* Empty *)
	{attribute 'hide'}
	bDiagBIT4						: BIT; 		(* Empty *)
	{attribute 'hide'}
	bDiagBIT5						: BIT; 		(* Empty *)
	{attribute 'hide'}
	bDiagBIT6						: BIT; 		(* Empty *)
	{attribute 'hide'}
	bDiagBIT7						: BIT; 		(* Empty *)
	{attribute 'hide'}
	bDiagBIT8						: BIT; 		(* Empty *)
	{attribute 'hide'}
	bDiagBIT9						: BIT; 		(* Empty *)
	{attribute 'hide'}
	bDiagBIT10						: BIT; 		(* Empty *)
	{attribute 'hide'}
	bDiagBIT11						: BIT; 		(* Empty *)
	{attribute 'hide'}
	bDiagBIT12						: BIT; 		(* Empty *)
	{attribute 'hide'}
	bDiagBIT13						: BIT; 		(* Empty *)
	{attribute 'hide'}
	bDiagBIT14						: BIT; 		(* Empty *)
	{attribute 'hide'}
	bDiagBIT15						: BIT; 		(* Empty *)
(* wInputs *)
	bIn_Restart						: BIT; 		(* .0 *)
	{attribute 'hide'}
	bInputBIT1						: BIT; 		(* Empty *)
	{attribute 'hide'}
	bInputBIT2						: BIT; 		(* Empty *)
	{attribute 'hide'}
	bInputBIT3						: BIT; 		(* Empty *)
	{attribute 'hide'}
	bInputBIT4						: BIT; 		(* Empty *)
	{attribute 'hide'}
	bInputBIT5						: BIT; 		(* Empty *)
	{attribute 'hide'}
	bInputBIT6						: BIT; 		(* Empty *)
	{attribute 'hide'}
	bInputBIT7						: BIT; 		(* Empty *)
	bIn_OPMODEIn1					: BIT; 		(* .8 *)
	bIn_OPMODEIn2					: BIT; 		(* .9 *)
	bIn_OPMODEIn3					: BIT; 		(* .10 *)
	bIn_OPMODEIn4					: BIT; 		(* .11 *)
	bIn_OPMODEIn5					: BIT; 		(* .12 *)
	bIn_OPMODEIn6					: BIT; 		(* .13 *)
	bIn_OPMODEIn7					: BIT; 		(* .14 *)
	bIn_OPMODEIn8					: BIT; 		(* .15 *)
(* wOutputs *)
	bOut_Error						: BIT; 		(* .0 *)
	{attribute 'hide'}
	bOutputBIT1						: BIT; 		(* Empty *)
	{attribute 'hide'}
	bOutputBIT2						: BIT; 		(* Empty *)
	{attribute 'hide'}
	bOutputBIT3						: BIT; 		(* Empty *)
	{attribute 'hide'}
	bOutputBIT4						: BIT; 		(* Empty *)
	{attribute 'hide'}
	bOutputBIT5						: BIT; 		(* Empty *)
	{attribute 'hide'}
	bOutputBIT6						: BIT; 		(* Empty *)
	{attribute 'hide'}
	bOutputBIT7						: BIT; 		(* Empty *)
	bOut_OPMODEOut1					: BIT; 		(* .8 *)
	bOut_OPMODEOut2					: BIT; 		(* .9 *)
	bOut_OPMODEOut3					: BIT; 		(* .10 *)
	bOut_OPMODEOut4					: BIT; 		(* .11 *)
	bOut_OPMODEOut5					: BIT; 		(* .12 *)
	bOut_OPMODEOut6					: BIT; 		(* .13 *)
	bOut_OPMODEOut7					: BIT; 		(* .14 *)
	bOut_OPMODEOut8					: BIT; 		(* .15 *)
END_STRUCT
END_TYPE

// ---- DUTs/FBs/FBStatus/ST_SAFETY_OR.TcDUT
TYPE ST_SAFETY_OR :
STRUCT
	{attribute 'hide'}
	BUnknown						: BYTE;
	BState							: BYTE;
(* wDiagnosis *)
	{attribute 'hide'}
	bDiagBIT0						: BIT; 		(* Empty *)
	{attribute 'hide'}
	bDiagBIT1						: BIT; 		(* Empty *)
	{attribute 'hide'}
	bDiagBIT2						: BIT; 		(* Empty *)
	{attribute 'hide'}
	bDiagBIT3						: BIT; 		(* Empty *)
	{attribute 'hide'}
	bDiagBIT4						: BIT; 		(* Empty *)
	{attribute 'hide'}
	bDiagBIT5						: BIT; 		(* Empty *)
	{attribute 'hide'}
	bDiagBIT6						: BIT; 		(* Empty *)
	{attribute 'hide'}
	bDiagBIT7						: BIT; 		(* Empty *)
	{attribute 'hide'}
	bDiagBIT8						: BIT; 		(* Empty *)
	{attribute 'hide'}
	bDiagBIT9						: BIT; 		(* Empty *)
	{attribute 'hide'}
	bDiagBIT10						: BIT; 		(* Empty *)
	{attribute 'hide'}
	bDiagBIT11						: BIT; 		(* Empty *)
	{attribute 'hide'}
	bDiagBIT12						: BIT; 		(* Empty *)
	{attribute 'hide'}
	bDiagBIT13						: BIT; 		(* Empty *)
	{attribute 'hide'}
	bDiagBIT14						: BIT; 		(* Empty *)
	{attribute 'hide'}
	bDiagBIT15						: BIT; 		(* Empty *)
(* wInputs *)
	{attribute 'hide'}
	bInputBIT0						: BIT; 		(* Empty *)
	{attribute 'hide'}
	bInputBIT1						: BIT; 		(* Empty *)
	{attribute 'hide'}
	bInputBIT2						: BIT; 		(* Empty *)
	{attribute 'hide'}
	bInputBIT3						: BIT; 		(* Empty *)
	{attribute 'hide'}
	bInputBIT4						: BIT; 		(* Empty *)
	{attribute 'hide'}
	bInputBIT5						: BIT; 		(* Empty *)
	{attribute 'hide'}
	bInputBIT6						: BIT; 		(* Empty *)
	{attribute 'hide'}
	bInputBIT7						: BIT; 		(* Empty *)
	bIn_ORIn1						: BOOL; 	(* .8 *)
	bIn_ORIn2						: BOOL; 	(* .9 *)
	bIn_ORIn3						: BOOL; 	(* .10 *)
	bIn_ORIn4						: BOOL; 	(* .11 *)
	bIn_ORIn5						: BOOL; 	(* .12 *)
	bIn_ORIn6						: BOOL; 	(* .13 *)
	bIn_ORIn7						: BOOL; 	(* .14 *)
	bIn_ORIn8						: BOOL; 	(* .15 *)
(* wOutputs *)
	bOut_OROut						: BOOL; 	(* .0 *)
	{attribute 'hide'}
	bOutputBIT1						: BIT; 		(* Empty *)
	{attribute 'hide'}
	bOutputBIT2						: BIT; 		(* Empty *)
	{attribute 'hide'}
	bOutputBIT3						: BIT; 		(* Empty *)
	{attribute 'hide'}
	bOutputBIT4						: BIT; 		(* Empty *)
	{attribute 'hide'}
	bOutputBIT5						: BIT; 		(* Empty *)
	{attribute 'hide'}
	bOutputBIT6						: BIT; 		(* Empty *)
	{attribute 'hide'}
	bOutputBIT7						: BIT; 		(* Empty *)
	{attribute 'hide'}
	bOutputBIT8						: BIT; 		(* Empty *)
	{attribute 'hide'}
	bOutputBIT9						: BIT; 		(* Empty *)
	{attribute 'hide'}
	bOutputBIT10					: BIT; 		(* Empty *)
	{attribute 'hide'}
	bOutputBIT11					: BIT; 		(* Empty *)
	{attribute 'hide'}
	bOutputBIT12					: BIT; 		(* Empty *)
	{attribute 'hide'}
	bOutputBIT13					: BIT; 		(* Empty *)
	{attribute 'hide'}
	bOutputBIT14					: BIT; 		(* Empty *)
	{attribute 'hide'}
	bOutputBIT15					: BIT; 		(* Empty *)
END_STRUCT
END_TYPE

// ---- DUTs/FBs/FBStatus/ST_SAFETY_RS.TcDUT
TYPE ST_SAFETY_RS :
STRUCT
	{attribute 'hide'}
	BUnknown						: BYTE;
	BState							: BYTE;
(* wDiagnosis *)
	{attribute 'hide'}
	bDiagBIT0						: BIT; 		(* Empty *)
	{attribute 'hide'}
	bDiagBIT1						: BIT; 		(* Empty *)
	{attribute 'hide'}
	bDiagBIT2						: BIT; 		(* Empty *)
	{attribute 'hide'}
	bDiagBIT3						: BIT; 		(* Empty *)
	{attribute 'hide'}
	bDiagBIT4						: BIT; 		(* Empty *)
	{attribute 'hide'}
	bDiagBIT5						: BIT; 		(* Empty *)
	{attribute 'hide'}
	bDiagBIT6						: BIT; 		(* Empty *)
	{attribute 'hide'}
	bDiagBIT7						: BIT; 		(* Empty *)
	{attribute 'hide'}
	bDiagBIT8						: BIT; 		(* Empty *)
	{attribute 'hide'}
	bDiagBIT9						: BIT; 		(* Empty *)
	{attribute 'hide'}
	bDiagBIT10						: BIT; 		(* Empty *)
	{attribute 'hide'}
	bDiagBIT11						: BIT; 		(* Empty *)
	{attribute 'hide'}
	bDiagBIT12						: BIT; 		(* Empty *)
	{attribute 'hide'}
	bDiagBIT13						: BIT; 		(* Empty *)
	{attribute 'hide'}
	bDiagBIT14						: BIT; 		(* Empty *)
	{attribute 'hide'}
	bDiagBIT15						: BIT; 		(* Empty *)
(* wInputs *)
	{attribute 'hide'}
	bInputBIT0						: BIT; 		(* Empty *)
	{attribute 'hide'}
	bInputBIT1						: BIT; 		(* Empty *)
	{attribute 'hide'}
	bInputBIT2						: BIT; 		(* Empty *)
	{attribute 'hide'}
	bInputBIT3						: BIT; 		(* Empty *)
	{attribute 'hide'}
	bInputBIT4						: BIT; 		(* Empty *)
	{attribute 'hide'}
	bInputBIT5						: BIT; 		(* Empty *)
	{attribute 'hide'}
	bInputBIT6						: BIT; 		(* Empty *)
	{attribute 'hide'}
	bInputBIT7						: BIT; 		(* Empty *)
	bIn_Reset						: BIT; 		(* .8 *)
	bIn_Set							: BIT; 		(* .9 *)
	{attribute 'hide'}
	bInputBIT10						: BIT; 		(* Empty *)
	{attribute 'hide'}
	bInputBIT11						: BIT; 		(* Empty *)
	{attribute 'hide'}
	bInputBIT12						: BIT; 		(* Empty *)
	{attribute 'hide'}
	bInputBIT13						: BIT; 		(* Empty *)
	{attribute 'hide'}
	bInputBIT14						: BIT; 		(* Empty *)
	{attribute 'hide'}
	bInputBIT15						: BIT; 		(* Empty *)
(* wOutputs *)
	{attribute 'hide'}
	bOut_OutputBIT0					: BIT; 		(* Empty *)
	bOut_RSOut						: BIT; 		(* .1 *)
	{attribute 'hide'}
	bOutputBIT2						: BIT; 		(* Empty *)
	{attribute 'hide'}
	bOutputBIT3						: BIT; 		(* Empty *)
	{attribute 'hide'}
	bOutputBIT4						: BIT; 		(* Empty *)
	{attribute 'hide'}
	bOutputBIT5						: BIT; 		(* Empty *)
	{attribute 'hide'}
	bOutputBIT6						: BIT; 		(* Empty *)
	{attribute 'hide'}
	bOutputBIT7						: BIT; 		(* Empty *)
	{attribute 'hide'}
	bOutputBIT8						: BIT; 		(* Empty *)
	{attribute 'hide'}
	bOutputBIT9						: BIT; 		(* Empty *)
	{attribute 'hide'}
	bOutputBIT10					: BIT; 		(* Empty *)
	{attribute 'hide'}
	bOutputBIT11					: BIT; 		(* Empty *)
	{attribute 'hide'}
	bOutputBIT12					: BIT; 		(* Empty *)
	{attribute 'hide'}
	bOutputBIT13					: BIT; 		(* Empty *)
	{attribute 'hide'}
	bOutputBIT14					: BIT; 		(* Empty *)
	{attribute 'hide'}
	bOutputBIT15					: BIT; 		(* Empty *)
END_STRUCT
END_TYPE

// ---- DUTs/FBs/FBStatus/ST_SAFETY_SR.TcDUT
TYPE ST_SAFETY_SR :
STRUCT
	{attribute 'hide'}
	BUnknown						: BYTE;
	BState							: BYTE;
(* wDiagnosis *)
	{attribute 'hide'}
	bDiagBIT0						: BIT; 		(* Empty *)
	{attribute 'hide'}
	bDiagBIT1						: BIT; 		(* Empty *)
	{attribute 'hide'}
	bDiagBIT2						: BIT; 		(* Empty *)
	{attribute 'hide'}
	bDiagBIT3						: BIT; 		(* Empty *)
	{attribute 'hide'}
	bDiagBIT4						: BIT; 		(* Empty *)
	{attribute 'hide'}
	bDiagBIT5						: BIT; 		(* Empty *)
	{attribute 'hide'}
	bDiagBIT6						: BIT; 		(* Empty *)
	{attribute 'hide'}
	bDiagBIT7						: BIT; 		(* Empty *)
	{attribute 'hide'}
	bDiagBIT8						: BIT; 		(* Empty *)
	{attribute 'hide'}
	bDiagBIT9						: BIT; 		(* Empty *)
	{attribute 'hide'}
	bDiagBIT10						: BIT; 		(* Empty *)
	{attribute 'hide'}
	bDiagBIT11						: BIT; 		(* Empty *)
	{attribute 'hide'}
	bDiagBIT12						: BIT; 		(* Empty *)
	{attribute 'hide'}
	bDiagBIT13						: BIT; 		(* Empty *)
	{attribute 'hide'}
	bDiagBIT14						: BIT; 		(* Empty *)
	{attribute 'hide'}
	bDiagBIT15						: BIT; 		(* Empty *)
(* wInputs *)
	{attribute 'hide'}
	bInputBIT0						: BIT; 		(* Empty *)
	{attribute 'hide'}
	bInputBIT1						: BIT; 		(* Empty *)
	{attribute 'hide'}
	bInputBIT2						: BIT; 		(* Empty *)
	{attribute 'hide'}
	bInputBIT3						: BIT; 		(* Empty *)
	{attribute 'hide'}
	bInputBIT4						: BIT; 		(* Empty *)
	{attribute 'hide'}
	bInputBIT5						: BIT; 		(* Empty *)
	{attribute 'hide'}
	bInputBIT6						: BIT; 		(* Empty *)
	{attribute 'hide'}
	bInputBIT7						: BIT; 		(* Empty *)
	bIn_Set							: BIT; 		(* .8 *)
	bIn_Reset						: BIT; 		(* .9 *)
	{attribute 'hide'}
	bInputBIT10						: BIT; 		(* Empty *)
	{attribute 'hide'}
	bInputBIT11						: BIT; 		(* Empty *)
	{attribute 'hide'}
	bInputBIT12						: BIT; 		(* Empty *)
	{attribute 'hide'}
	bInputBIT13						: BIT; 		(* Empty *)
	{attribute 'hide'}
	bInputBIT14						: BIT; 		(* Empty *)
	{attribute 'hide'}
	bInputBIT15						: BIT; 		(* Empty *)
(* wOutputs *)
	{attribute 'hide'}
	bOutputBIT0						: BIT; 		(* Empty *)
	bOut_SROut						: BIT; 		(* .1 *)
	{attribute 'hide'}
	bOutputBIT2						: BIT; 		(* Empty *)
	{attribute 'hide'}
	bOutputBIT3						: BIT; 		(* Empty *)
	{attribute 'hide'}
	bOutputBIT4						: BIT; 		(* Empty *)
	{attribute 'hide'}
	bOutputBIT5						: BIT; 		(* Empty *)
	{attribute 'hide'}
	bOutputBIT6						: BIT; 		(* Empty *)
	{attribute 'hide'}
	bOutputBIT7						: BIT; 		(* Empty *)
	{attribute 'hide'}
	bOutputBIT8						: BIT; 		(* Empty *)
	{attribute 'hide'}
	bOutputBIT9						: BIT; 		(* Empty *)
	{attribute 'hide'}
	bOutputBIT10					: BIT; 		(* Empty *)
	{attribute 'hide'}
	bOutputBIT11					: BIT; 		(* Empty *)
	{attribute 'hide'}
	bOutputBIT12					: BIT; 		(* Empty *)
	{attribute 'hide'}
	bOutputBIT13					: BIT; 		(* Empty *)
	{attribute 'hide'}
	bOutputBIT14					: BIT; 		(* Empty *)
	{attribute 'hide'}
	bOutputBIT15					: BIT; 		(* Empty *)
END_STRUCT
END_TYPE

// ---- DUTs/FBs/FBStatus/ST_SAFETY_TOF.TcDUT
TYPE ST_SAFETY_TOF :
STRUCT
	{attribute 'hide'}
	BUnknown						: BYTE;
	BState							: BYTE;
(* wDiagnosis *)
	{attribute 'hide'}
	bDiagBIT0						: BIT; 		(* Empty *)
	{attribute 'hide'}
	bDiagBIT1						: BIT; 		(* Empty *)
	{attribute 'hide'}
	bDiagBIT2						: BIT; 		(* Empty *)
	{attribute 'hide'}
	bDiagBIT3						: BIT; 		(* Empty *)
	{attribute 'hide'}
	bDiagBIT4						: BIT; 		(* Empty *)
	{attribute 'hide'}
	bDiagBIT5						: BIT; 		(* Empty *)
	{attribute 'hide'}
	bDiagBIT6						: BIT; 		(* Empty *)
	{attribute 'hide'}
	bDiagBIT7						: BIT; 		(* Empty *)
	{attribute 'hide'}
	bDiagBIT8						: BIT; 		(* Empty *)
	{attribute 'hide'}
	bDiagBIT9						: BIT; 		(* Empty *)
	{attribute 'hide'}
	bDiagBIT10						: BIT; 		(* Empty *)
	{attribute 'hide'}
	bDiagBIT11						: BIT; 		(* Empty *)
	{attribute 'hide'}
	bDiagBIT12						: BIT; 		(* Empty *)
	{attribute 'hide'}
	bDiagBIT13						: BIT; 		(* Empty *)
	{attribute 'hide'}
	bDiagBIT14						: BIT; 		(* Empty *)
	{attribute 'hide'}
	bDiagBIT15						: BIT; 		(* Empty *)
(* wInputs *)
	{attribute 'hide'}
	bInputBIT0						: BIT; 		(* Empty *)
	{attribute 'hide'}
	bInputBIT1						: BIT; 		(* Empty *)
	{attribute 'hide'}
	bInputBIT2						: BIT; 		(* Empty *)
	{attribute 'hide'}
	bInputBIT3						: BIT; 		(* Empty *)
	{attribute 'hide'}
	bInputBIT4						: BIT; 		(* Empty *)
	{attribute 'hide'}
	bInputBIT5						: BIT; 		(* Empty *)
	{attribute 'hide'}
	bInputBIT6						: BIT; 		(* Empty *)
	{attribute 'hide'}
	bInputBIT7						: BIT; 		(* Empty *)
	bIn_TofIn						: BIT; 		(* .8 *)
	{attribute 'hide'}
	bInputBIT9						: BIT; 		(* Empty *)
	{attribute 'hide'}
	bInputBIT10						: BIT; 		(* Empty *)
	{attribute 'hide'}
	bInputBIT11						: BIT; 		(* Empty *)
	{attribute 'hide'}
	bInputBIT12						: BIT; 		(* Empty *)
	{attribute 'hide'}
	bInputBIT13						: BIT; 		(* Empty *)
	{attribute 'hide'}
	bInputBIT14						: BIT; 		(* Empty *)
	{attribute 'hide'}
	bInputBIT15						: BIT; 		(* Empty *)
(* wOutputs *)
	{attribute 'hide'}
	bOutputBIT0						: BIT; 		(* Empty *)
	bOut_TofOut						: BIT; 		(* .1 *)
	{attribute 'hide'}
	bOutputBIT2						: BIT; 		(* Empty *)
	{attribute 'hide'}
	bOutputBIT3						: BIT; 		(* Empty *)
	{attribute 'hide'}
	bOutputBIT4						: BIT; 		(* Empty *)
	{attribute 'hide'}
	bOutputBIT5						: BIT; 		(* Empty *)
	{attribute 'hide'}
	bOutputBIT6						: BIT; 		(* Empty *)
	{attribute 'hide'}
	bOutputBIT7						: BIT; 		(* Empty *)
	{attribute 'hide'}
	bOutputBIT8						: BIT; 		(* Empty *)
	{attribute 'hide'}
	bOutputBIT9						: BIT; 		(* Empty *)
	{attribute 'hide'}
	bOutputBIT10					: BIT; 		(* Empty *)
	{attribute 'hide'}
	bOutputBIT11					: BIT; 		(* Empty *)
	{attribute 'hide'}
	bOutputBIT12					: BIT; 		(* Empty *)
	{attribute 'hide'}
	bOutputBIT13					: BIT; 		(* Empty *)
	{attribute 'hide'}
	bOutputBIT14					: BIT; 		(* Empty *)
	{attribute 'hide'}
	bOutputBIT15					: BIT; 		(* Empty *)
END_STRUCT
END_TYPE

// ---- DUTs/FBs/FBStatus/ST_SAFETY_TON.TcDUT
TYPE ST_SAFETY_TON :
STRUCT
	{attribute 'hide'}
	BUnknown						: BYTE;
	BState							: BYTE;
(* wDiagnosis *)
	{attribute 'hide'}
	bDiagBIT0						: BIT; 		(* Empty *)
	{attribute 'hide'}
	bDiagBIT1						: BIT; 		(* Empty *)
	{attribute 'hide'}
	bDiagBIT2						: BIT; 		(* Empty *)
	{attribute 'hide'}
	bDiagBIT3						: BIT; 		(* Empty *)
	{attribute 'hide'}
	bDiagBIT4						: BIT; 		(* Empty *)
	{attribute 'hide'}
	bDiagBIT5						: BIT; 		(* Empty *)
	{attribute 'hide'}
	bDiagBIT6						: BIT; 		(* Empty *)
	{attribute 'hide'}
	bDiagBIT7						: BIT; 		(* Empty *)
	{attribute 'hide'}
	bDiagBIT8						: BIT; 		(* Empty *)
	{attribute 'hide'}
	bDiagBIT9						: BIT; 		(* Empty *)
	{attribute 'hide'}
	bDiagBIT10						: BIT; 		(* Empty *)
	{attribute 'hide'}
	bDiagBIT11						: BIT; 		(* Empty *)
	{attribute 'hide'}
	bDiagBIT12						: BIT; 		(* Empty *)
	{attribute 'hide'}
	bDiagBIT13						: BIT; 		(* Empty *)
	{attribute 'hide'}
	bDiagBIT14						: BIT; 		(* Empty *)
	{attribute 'hide'}
	bDiagBIT15						: BIT; 		(* Empty *)
(* wInputs *)
	{attribute 'hide'}
	bInputBIT0						: BIT; 		(* Empty *)
	{attribute 'hide'}
	bInputBIT1						: BIT; 		(* Empty *)
	{attribute 'hide'}
	bInputBIT2						: BIT; 		(* Empty *)
	{attribute 'hide'}
	bInputBIT3						: BIT; 		(* Empty *)
	{attribute 'hide'}
	bInputBIT4						: BIT; 		(* Empty *)
	{attribute 'hide'}
	bInputBIT5						: BIT; 		(* Empty *)
	{attribute 'hide'}
	bInputBIT6						: BIT; 		(* Empty *)
	{attribute 'hide'}
	bInputBIT7						: BIT; 		(* Empty *)
	bIn_TonIn						: BIT; 		(* .8 *)
	bInputBIT9						: BIT; 		(* Empty *)
	{attribute 'hide'}
	bInputBIT10						: BIT; 		(* Empty *)
	{attribute 'hide'}
	bInputBIT11						: BIT; 		(* Empty *)
	{attribute 'hide'}
	bInputBIT12						: BIT; 		(* Empty *)
	{attribute 'hide'}
	bInputBIT13						: BIT; 		(* Empty *)
	{attribute 'hide'}
	bInputBIT14						: BIT; 		(* Empty *)
	{attribute 'hide'}
	bInputBIT15						: BIT; 		(* Empty *)
(* wOutputs *)
	{attribute 'hide'}
	bOutputBIT0						: BIT; 		(* Empty *)
	bOut_TonOut						: BIT; 		(* .1 *)
	{attribute 'hide'}
	bOutputBIT2						: BIT; 		(* Empty *)
	{attribute 'hide'}
	bOutputBIT3						: BIT; 		(* Empty *)
	{attribute 'hide'}
	bOutputBIT4						: BIT; 		(* Empty *)
	{attribute 'hide'}
	bOutputBIT5						: BIT; 		(* Empty *)
	{attribute 'hide'}
	bOutputBIT6						: BIT; 		(* Empty *)
	{attribute 'hide'}
	bOutputBIT7						: BIT; 		(* Empty *)
	{attribute 'hide'}
	bOutputBIT8						: BIT; 		(* Empty *)
	{attribute 'hide'}
	bOutputBIT9						: BIT; 		(* Empty *)
	{attribute 'hide'}
	bOutputBIT10					: BIT; 		(* Empty *)
	{attribute 'hide'}
	bOutputBIT11					: BIT; 		(* Empty *)
	{attribute 'hide'}
	bOutputBIT12					: BIT; 		(* Empty *)
	{attribute 'hide'}
	bOutputBIT13					: BIT; 		(* Empty *)
	{attribute 'hide'}
	bOutputBIT14					: BIT; 		(* Empty *)
	{attribute 'hide'}
	bOutputBIT15					: BIT; 		(* Empty *)
END_STRUCT
END_TYPE

// ---- DUTs/FBs/FBStatus/ST_SAFETY_TWOHAND.TcDUT
TYPE ST_SAFETY_TWOHAND :
STRUCT
	{attribute 'hide'}
	BUnknown						: BYTE;
	BState							: BYTE;
(* wDiagnosis *)
	bDiag_DiscErrorTWOHANDIn1_2		: BIT;		(*	Discrepancy error input group 1	*)
	bDiag_DiscErrorTWOHANDIn3_4		: BIT;		(*	Discrepancy error input group 2	*)
	bDiag_DiscErrorTWOHANDIn1_2_3_4	: BIT;		(*	Discrepancy error between the two input groups 	*)
	{attribute 'hide'}
	bDiagBIT3						: BIT; 		(* Empty *)
	{attribute 'hide'}
	bDiagBIT4						: BIT; 		(* Empty *)
	{attribute 'hide'}
	bDiagBIT5						: BIT; 		(* Empty *)
	bDiag_TwoHandError				: BIT;		(* Two-hand error	*)
	{attribute 'hide'}
	bDiagBIT7						: BIT; 		(* Empty *)
	{attribute 'hide'}
	bDiagBIT8						: BIT; 		(* Empty *)
	{attribute 'hide'}
	bDiagBIT9						: BIT; 		(* Empty *)
	{attribute 'hide'}
	bDiagBIT10						: BIT; 		(* Empty *)
	{attribute 'hide'}
	bDiagBIT11						: BIT; 		(* Empty *)
	{attribute 'hide'}
	bDiagBIT12						: BIT; 		(* Empty *)
	{attribute 'hide'}
	bDiagBIT13						: BIT; 		(* Empty *)
	{attribute 'hide'}
	bDiagBIT14						: BIT; 		(* Empty *)
	{attribute 'hide'}
	bDiagBIT15						: BIT; 		(* Empty *)
(* wInputs *)
	{attribute 'hide'}
	bInputBIT0						: BIT; 		(* Empty *)
	{attribute 'hide'}
	bInputBIT1						: BIT; 		(* Empty *)
	{attribute 'hide'}
	bInputBIT2						: BIT; 		(* Empty *)
	{attribute 'hide'}
	bInputBIT3						: BIT; 		(* Empty *)
	{attribute 'hide'}
	bInputBIT4						: BIT; 		(* Empty *)
	{attribute 'hide'}
	bInputBIT5						: BIT; 		(* Empty *)
	{attribute 'hide'}
	bInputBIT6						: BIT; 		(* Empty *)
	{attribute 'hide'}
	bInputBIT7						: BIT; 		(* Empty *)
	bIn_TWOHANDIn1					: BIT; 		(* .8 *)
	bIn_TWOHANDIn2					: BIT; 		(* .9 *)
	bIn_TWOHANDIn3					: BIT; 		(* .10 *)
	bIn_TWOHANDIn4					: BIT; 		(* .11 *)
	{attribute 'hide'}
	bInputBIT12						: BIT; 		(* Empty *)
	{attribute 'hide'}
	bInputBIT13						: BIT; 		(* Empty *)
	{attribute 'hide'}
	bInputBIT14						: BIT; 		(* Empty *)
	{attribute 'hide'}
	bInputBIT15						: BIT; 		(* Empty *)
(* wOutputs *)
	bOut_Error						: BIT; 		(* .0 *)
	bOut_TWOHANDOut					: BIT; 		(* .1 *)
	{attribute 'hide'}
	bOutputBIT2						: BIT; 		(* Empty *)
	{attribute 'hide'}
	bOutputBIT3						: BIT; 		(* Empty *)
	{attribute 'hide'}
	bOutputBIT4						: BIT; 		(* Empty *)
	{attribute 'hide'}
	bOutputBIT5						: BIT; 		(* Empty *)
	{attribute 'hide'}
	bOutputBIT6						: BIT; 		(* Empty *)
	{attribute 'hide'}
	bOutputBIT7						: BIT; 		(* Empty *)
	{attribute 'hide'}
	bOutputBIT8						: BIT; 		(* Empty *)
	{attribute 'hide'}
	bOutputBIT9						: BIT; 		(* Empty *)
	{attribute 'hide'}
	bOutputBIT10					: BIT; 		(* Empty *)
	{attribute 'hide'}
	bOutputBIT11					: BIT; 		(* Empty *)
	{attribute 'hide'}
	bOutputBIT12					: BIT; 		(* Empty *)
	{attribute 'hide'}
	bOutputBIT13					: BIT; 		(* Empty *)
	{attribute 'hide'}
	bOutputBIT14					: BIT; 		(* Empty *)
	{attribute 'hide'}
	bOutputBIT15					: BIT; 		(* Empty *)
END_STRUCT
END_TYPE

// ---- DUTs/FBs/ST_SAFETY_FBAND.TcDUT
TYPE ST_SAFETY_FBAND:
STRUCT
	uStatus							: U_SAFETY_AND; 		(* Typ zalezny od bloku *)
	eState							: E_SAFETY_FBState;		(* Enum ze statusem bloku *)
	bGeneralError					: BOOL; 				(* Gdy wystapi chociaz jeden Error *)
END_STRUCT
END_TYPE

// ---- DUTs/FBs/ST_SAFETY_FBCONNECTIONSHUTDOWN.TcDUT
TYPE ST_SAFETY_FBCONNECTIONSHUTDOWN:
STRUCT
	uStatus							: U_SAFETY_CONNECTIONSHUTDOWN; 		(* Typ zalezny od bloku *)
	eState							: E_SAFETY_FBStateCS;				(* Enum ze statusem bloku *)
	bGeneralError					: BOOL; 							(* Gdy wystapi chociaz jeden Error *)	
END_STRUCT
END_TYPE

// ---- DUTs/FBs/ST_SAFETY_FBDECOUPLE.TcDUT
TYPE ST_SAFETY_FBDECOUPLE:
STRUCT
	uStatus							: U_SAFETY_DECOUPLE; 		(* Typ zalezny od bloku *)
	eState							: E_SAFETY_FBState;			(* Enum ze statusem bloku *)
	bGeneralError					: BOOL; 					(* Gdy wystapi chociaz jeden Error *)
END_STRUCT
END_TYPE

// ---- DUTs/FBs/ST_SAFETY_FBEDM.TcDUT
TYPE ST_SAFETY_FBEDM:
STRUCT
	uStatus							: U_SAFETY_EDM; 		(* Typ zalezny od bloku *)
	eState							: E_SAFETY_FBState;		(* Enum ze statusem bloku *)
	bGeneralError					: BOOL; 				(* Gdy wystapi chociaz jeden Error *)
END_STRUCT
END_TYPE

// ---- DUTs/FBs/ST_SAFETY_FBESTOP.TcDUT
TYPE ST_SAFETY_FBESTOP:
STRUCT
	uStatus							: U_SAFETY_ESTOP; 		(* Typ zalezny od bloku *)
	eState							: E_SAFETY_FBState;		(* Enum ze statusem bloku *)
	bGeneralError					: BOOL; 				(* Gdy wystapi chociaz jeden Error *)
END_STRUCT
END_TYPE

// ---- DUTs/FBs/ST_SAFETY_FBMON.TcDUT
TYPE ST_SAFETY_FBMON:
STRUCT
	uStatus							: U_SAFETY_MON; 		(* Typ zalezny od bloku *)
	eState							: E_SAFETY_FBState;		(* Enum ze statusem bloku *)
	bGeneralError					: BOOL; 				(* Gdy wystapi chociaz jeden Error *)
END_STRUCT
END_TYPE

// ---- DUTs/FBs/ST_SAFETY_FBMUTING.TcDUT
TYPE ST_SAFETY_FBMUTING:
STRUCT
	uStatus							: U_SAFETY_MUTING; 				(* Typ zalezny od bloku *)
	eState							: E_SAFETY_FBStateMUTING;		(* Enum ze statusem bloku *)
	bGeneralError					: BOOL; 						(* Gdy wystapi chociaz jeden Error *)
END_STRUCT
END_TYPE

// ---- DUTs/FBs/ST_SAFETY_FBOPMODE.TcDUT
TYPE ST_SAFETY_FBOPMODE:
STRUCT
	uStatus							: U_SAFETY_OPMODE; 		(* Typ zalezny od bloku *)
	eState							: E_SAFETY_FBState;		(* Enum ze statusem bloku *)
	bGeneralError					: BOOL; 				(* Gdy wystapi chociaz jeden Error *)
END_STRUCT
END_TYPE

// ---- DUTs/FBs/ST_SAFETY_FBOR.TcDUT
TYPE ST_SAFETY_FBOR:
STRUCT
	uStatus							: U_SAFETY_OR; 			(* Typ zalezny od bloku *)
	eState							: E_SAFETY_FBState;		(* Enum ze statusem bloku *)
	bGeneralError					: BOOL; 				(* Gdy wystapi chociaz jeden Error *)
END_STRUCT
END_TYPE

// ---- DUTs/FBs/ST_SAFETY_FBRS.TcDUT
TYPE ST_SAFETY_FBRS:
STRUCT
	uStatus							: U_SAFETY_RS; 					(* Typ zalezny od bloku *)
	eState							: E_SAFETY_FBStateSetReset;		(* Enum ze statusem bloku *)
	bGeneralError					: BOOL; 						(* Gdy wystapi chociaz jeden Error *)
END_STRUCT
END_TYPE

// ---- DUTs/FBs/ST_SAFETY_FBSR.TcDUT
TYPE ST_SAFETY_FBSR:
STRUCT
	uStatus							: U_SAFETY_SR; 					(* Typ zalezny od bloku *)
	eState							: E_SAFETY_FBStateSetReset;		(* Enum ze statusem bloku *)
	bGeneralError					: BOOL; 						(* Gdy wystapi chociaz jeden Error *)
END_STRUCT
END_TYPE

// ---- DUTs/FBs/ST_SAFETY_FBTOF.TcDUT
TYPE ST_SAFETY_FBTOF:
STRUCT
	uStatus							: U_SAFETY_TOF; 				(* Typ zalezny od bloku *)
	eState							: E_SAFETY_FBStateTimer;		(* Enum ze statusem bloku *)
	bGeneralError					: BOOL; 						(* Gdy wystapi chociaz jeden Error *)
END_STRUCT
END_TYPE

// ---- DUTs/FBs/ST_SAFETY_FBTON.TcDUT
TYPE ST_SAFETY_FBTON:
STRUCT
	uStatus							: U_SAFETY_TON; 				(* Typ zalezny od bloku *)
	eState							: E_SAFETY_FBStateTimer;		(* Enum ze statusem bloku *)
	bGeneralError					: BOOL; 						(* Gdy wystapi chociaz jeden Error *)
END_STRUCT
END_TYPE

// ---- DUTs/FBs/ST_SAFETY_FBTWOHAND.TcDUT
TYPE ST_SAFETY_FBTWOHAND:
STRUCT
	uStatus							: U_SAFETY_TWOHAND; 	(* Typ zalezny od bloku *)
	eState							: E_SAFETY_FBState;		(* Enum ze statusem bloku *)
	bGeneralError					: BOOL; 				(* Gdy wystapi chociaz jeden Error *)
END_STRUCT
END_TYPE

// ---- DUTs/FBs/Unions/U_SAFETY_AND.TcDUT
TYPE U_SAFETY_AND :
UNION
	stStatusWords					: ST_SAFETY_FBStatus;		(* BUnknown, BState, wDiagnosis, wInputs, wOutputs - takie same dla wszystkich FB *)
	stStatus						: ST_SAFETY_AND; 			(* Rozbite na Bity - inne dla kazdego bloku*)
END_UNION
END_TYPE

// ---- DUTs/FBs/Unions/U_SAFETY_CONNECTIONSHUTDOWN.TcDUT
TYPE U_SAFETY_CONNECTIONSHUTDOWN :
UNION
	stStatusWords					: ST_SAFETY_FBStatus;				(* BUnknown, BState, wDiagnosis, wInputs, wOutputs - takie same dla wszystkich FB *)
	stStatus						: ST_SAFETY_CONNECTIONSHUTDOWN; 	(* Rozbite na Bity - inne dla kazdego bloku*)
END_UNION
END_TYPE

// ---- DUTs/FBs/Unions/U_SAFETY_DECOUPLE.TcDUT
TYPE U_SAFETY_DECOUPLE :
UNION
	stStatusWords					: ST_SAFETY_FBStatus;			(* BUnknown, BState, wDiagnosis, wInputs, wOutputs - takie same dla wszystkich FB *)
	stStatus						: ST_SAFETY_DECOUPLE; 			(* Rozbite na Bity - inne dla kazdego bloku*)
END_UNION
END_TYPE

// ---- DUTs/FBs/Unions/U_SAFETY_EDM.TcDUT
TYPE U_SAFETY_EDM :
UNION
	stStatusWords					: ST_SAFETY_FBStatus;			(* BUnknown, BState, wDiagnosis, wInputs, wOutputs - takie same dla wszystkich FB *)
	stStatus						: ST_SAFETY_EDM; 				(* Rozbite na Bity - inne dla kazdego bloku*)
END_UNION
END_TYPE

// ---- DUTs/FBs/Unions/U_SAFETY_ESTOP.TcDUT
TYPE U_SAFETY_ESTOP :
UNION
	stStatusWords					: ST_SAFETY_FBStatus;		(* BUnknown, BState, wDiagnosis, wInputs, wOutputs - takie same dla wszystkich FB *)
	stStatus						: ST_SAFETY_ESTOP; 			(* Rozbite na Bity - inne dla kazdego bloku*)
END_UNION
END_TYPE

// ---- DUTs/FBs/Unions/U_SAFETY_MON.TcDUT
TYPE U_SAFETY_MON :
UNION
	stStatusWords					: ST_SAFETY_FBStatus;		(* BUnknown, BState, wDiagnosis, wInputs, wOutputs - takie same dla wszystkich FB *)
	stStatus						: ST_SAFETY_MON; 			(* Rozbite na Bity - inne dla kazdego bloku*)
END_UNION
END_TYPE

// ---- DUTs/FBs/Unions/U_SAFETY_MUTING.TcDUT
TYPE U_SAFETY_MUTING :
UNION
	stStatusWords					: ST_SAFETY_FBStatus;			(* BUnknown, BState, wDiagnosis, wInputs, wOutputs - takie same dla wszystkich FB *)
	stStatus						: ST_SAFETY_MUTING; 			(* Rozbite na Bity - inne dla kazdego bloku*)
END_UNION
END_TYPE

// ---- DUTs/FBs/Unions/U_SAFETY_OPMODE.TcDUT
TYPE U_SAFETY_OPMODE :
UNION
	stStatusWords					: ST_SAFETY_FBStatus;			(* BUnknown, BState, wDiagnosis, wInputs, wOutputs - takie same dla wszystkich FB *)
	stStatus						: ST_SAFETY_OPMODE; 			(* Rozbite na Bity - inne dla kazdego bloku*)
END_UNION
END_TYPE

// ---- DUTs/FBs/Unions/U_SAFETY_OR.TcDUT
TYPE U_SAFETY_OR :
UNION
	stStatusWords					: ST_SAFETY_FBStatus;			(* BUnknown, BState, wDiagnosis, wInputs, wOutputs - takie same dla wszystkich FB *)
	stStatus						: ST_SAFETY_OR; 				(* Rozbite na Bity - inne dla kazdego bloku*)
END_UNION
END_TYPE

// ---- DUTs/FBs/Unions/U_SAFETY_RS.TcDUT
TYPE U_SAFETY_RS :
UNION
	stStatusWords					: ST_SAFETY_FBStatus;			(* BUnknown, BState, wDiagnosis, wInputs, wOutputs - takie same dla wszystkich FB *)
	stStatus						: ST_SAFETY_RS; 				(* Rozbite na Bity - inne dla kazdego bloku*)
END_UNION
END_TYPE

// ---- DUTs/FBs/Unions/U_SAFETY_SR.TcDUT
TYPE U_SAFETY_SR :
UNION
	stStatusWords					: ST_SAFETY_FBStatus;			(* BUnknown, BState, wDiagnosis, wInputs, wOutputs - takie same dla wszystkich FB *)
	stStatus						: ST_SAFETY_SR; 				(* Rozbite na Bity - inne dla kazdego bloku*)
END_UNION
END_TYPE

// ---- DUTs/FBs/Unions/U_SAFETY_TOF.TcDUT
TYPE U_SAFETY_TOF :
UNION
	stStatusWords					: ST_SAFETY_FBStatus;			(* BUnknown, BState, wDiagnosis, wInputs, wOutputs - takie same dla wszystkich FB *)
	stStatus						: ST_SAFETY_TOF; 				(* Rozbite na Bity - inne dla kazdego bloku*)
END_UNION
END_TYPE

// ---- DUTs/FBs/Unions/U_SAFETY_TON.TcDUT
TYPE U_SAFETY_TON :
UNION
	stStatusWords					: ST_SAFETY_FBStatus;			(* BUnknown, BState, wDiagnosis, wInputs, wOutputs - takie same dla wszystkich FB *)
	stStatus						: ST_SAFETY_TON;				(* Rozbite na Bity - inne dla kazdego bloku*)
END_UNION
END_TYPE

// ---- DUTs/FBs/Unions/U_SAFETY_TWOHAND.TcDUT
TYPE U_SAFETY_TWOHAND :
UNION
	stStatusWords					: ST_SAFETY_FBStatus;			(* BUnknown, BState, wDiagnosis, wInputs, wOutputs - takie same dla wszystkich FB *)
	stStatus						: ST_SAFETY_TWOHAND;			(* Rozbite na Bity - inne dla kazdego bloku*)
END_UNION
END_TYPE

// ---- DUTs/HW/E_AX580x_ERROR.TcDUT
// CoE object 0xFA82
TYPE E_AX580x_ERROR :
(	
	eAX580x_ERROR_FAULT_MAXT_C1		 					:= 16#0001,	// The temperature has exceeded the maximum permissible temperature (µC1).
	eAX580x_ERROR_FAULT_MAXT_C2			 				:= 16#0002,	// The temperature has exceeded the maximum permissible temperature (µC2).
	eAX580x_ERROR_FAULT_MINT_C1						 	:= 16#0003,	// The temperature has fallen below the minimum permissible temperature (µC1).
	eAX580x_ERROR_FAULT_MINT_C2 						:= 16#0004,	// The temperature has fallen below the minimum permissible temperature (µC2).
	eAX580x_ERROR_HW_ERR_MAX_VCC_C1						:= 16#0101,	// The maximum supply voltage was exceeded (3.3 V).
	eAX580x_ERROR_HW_ERR_MAX_VCC_C2					 	:= 16#0102,	// The maximum supply voltage was exceeded (3.3 V).
	eAX580x_ERROR_HW_ERR_MIN_VCC_C1			 			:= 16#0103,	// The supply voltage fell below the minimum value (3.3 V)
	eAX580x_ERROR_HW_ERR_MIN_VCC_C2						:= 16#0104,	// The supply voltage fell below the minimum value (3.3 V)
	eAX580x_ERROR_FAULT_MCTC1_TO						:= 16#0201,	// The MCTests of µC1 were not carried out completely within the specified time
	eAX580x_ERROR_FAULT_MCTC2_TO						:= 16#0202,	// The MCTests of µC2 were not carried out completely within the specified time
	eAX580x_ERROR_FAULT_TIMER_C1			 			:= 16#0203,	// The global timer was not updated in time.
	eAX580x_ERROR_FAULT_TIMER_C2						:= 16#0204,	// The global timer was not updated in time.
	eAX580x_ERROR_FAULT_TS_WDG_TO_C1					:= 16#020C,	// The TwinSAFE module was not called within the watchdog time.
	eAX580x_ERROR_FAULT_TS_WDG_TO_C2 					:= 16#020D,	// The TwinSAFE module was not called within the watchdog time.
	eAX580x_ERROR_FAULT_RESET_MC1 	 					:= 16#020E,	// A reset has occurred in the operation of the controller for µC1. µC2 was not reset thereby.
	eAX580x_ERROR_FAULT_SERCOMC2						:= 16#0300,	// an error occurred in the SerComP24C2 module during data transmission
	eAX580x_ERROR_FAULT_SERCOM1							:= 16#401,	// an error occurred in the SerComP24C1 module during data transmission
	eAX580x_ERROR_FAULT_SERCOM2							:= 16#402,	// an error occurred in the SerComP24C1 module during data transmission
	eAX580x_ERROR_FAULT_SERCOM3							:= 16#403,	// an error occurred in the SerComP24C1 module during data transmission
	eAX580x_ERROR_FAULT_SERCOM4							:= 16#404,	// an error occurred in the SerComP24C1 module during data transmission
	eAX580x_ERROR_FAULT_SERCOM5							:= 16#405,	// an error occurred in the SerComP24C1 module during data transmission
	eAX580x_ERROR_FAULT_SERCOM6							:= 16#406,	// an error occurred in the SerComP24C1 module during data transmission
	eAX580x_ERROR_FAULT_SERCOM7							:= 16#407,	// an error occurred in the SerComP24C1 module during data transmission
	eAX580x_ERROR_FAULT_SERCOM8							:= 16#408,	// an error occurred in the SerComP24C1 module during data transmission
	eAX580x_ERROR_FAULT_SERCOM9							:= 16#409,	// an error occurred in the SerComP24C1 module during data transmission
	eAX580x_ERROR_FAULT_SERCOM10 						:= 16#40A,	// an error occurred in the SerComP24C1 module during data transmission
	eAX580x_ERROR_FAULT_SERCOM11 						:= 16#40B,	// an error occurred in the SerComP24C1 module during data transmission
	eAX580x_ERROR_FAULT_TEMPSENSOR1						:= 16#501,	// Error in the communication with one of the temperature sensors
	eAX580x_ERROR_FAULT_TEMPSENSOR2 					:= 16#502,	// Error in the communication with one of the temperature sensors
	eAX580x_ERROR_FAULT_TEMPSENSOR3						:= 16#503,	// Error in the communication with one of the temperature sensors
	eAX580x_ERROR_FAULT_TEMPSENSOR4						:= 16#504,	// Error in the communication with one of the temperature sensors
	eAX580x_ERROR_FAULT_TEMPSENSOR5						:= 16#505,	// Error in the communication with one of the temperature sensors
	eAX580x_ERROR_FAULT_TEMPSENSOR6						:= 16#506,	// Error in the communication with one of the temperature sensors
	eAX580x_ERROR_FAULT_TEMPSENSOR7						:= 16#507,	// Error in the communication with one of the temperature sensors
	eAX580x_ERROR_FAULT_OUTPUTCOMPARE					:= 16#0601,	// The values output by µC1 and µC2 differ.
	eAX580x_ERROR_FAULT_OUTPUTCOMPAREC2			 		:= 16#0602,	// The values output by µC1 and µC2 differ.
	eAX580x_ERROR_HW_ERR_MIN_VCC_FPGA					:= 16#0700,	// The FPGA supply voltage fell below the minimum value (5 V).
	eAX580x_ERROR_HW_ERR_MAX_VCC_FPGA					:= 16#0701,	// The FPGA supply voltage exceeded the maximum value (5 V).
	eAX580x_ERROR_FAULT_FEEDBACK_C1						:= 16#0710,	// An error was detected in the feedback channels of µC1.
	eAX580x_ERROR_FAULT_FEEDBACK_C2						:= 16#0711,	// An error was detected in the feedback channels of µC2.
	eAX580x_ERROR_FAULT_Parameter_C1					:= 16#0720,	// General parameter error µC1 
	eAX580x_ERROR_FAULT_Parameter_C2					:= 16#0721,	// General parameter error µC2 
	eAX580x_ERROR_FAULT_Parameter_C1_DRIVE_PROFILE		:= 16#0722,	// Parameter: unknown parameter index µC1 drive profile
	eAX580x_ERROR_FAULT_Parameter_C1_VENDOR_SPECIFIC	:= 16#0723,	// Parameter: unknown parameter index µC1 vendor-specific.
	eAX580x_ERROR_FAULT_Parameter_C2_DRIVE_PROFILE		:= 16#0724,	// Parameter: unknown parameter index µC2 drive profile.
	eAX580x_ERROR_FAULT_Parameter_C2_VENDOR_SPECIFIC	:= 16#0725,	// Parameter: unknown parameter index µC2 vendor-specific.
	eAX580x_ERROR_FAULT_PDO_MAPPING_FSOE_COMMAND 		:= 16#0726,	// PDO mapping axis 1/2: FSOE COMMAND error.
	eAX580x_ERROR_FAULT_PDO_MAPPING_LENGTH				:= 16#0727,	// PDO mapping axis 1: Length_Error 
	eAX580x_ERROR_FAULT_PDO_MAPPING_STO_K1				:= 16#0728,	// PDO mapping axis 1: STO error 
	eAX580x_ERROR_FAULT_PDO_MAPPING_SS1_1_K1			:= 16#0729,	// PDO mapping axis 1: Error SS1_1 
	eAX580x_ERROR_FAULT_PDO_MAPPING_SS2_1_K1			:= 16#072A,	// PDO mapping axis 1: Error SS2_1 
	eAX580x_ERROR_FAULT_PDO_MAPPING_SOS_1_K1			:= 16#072B,	// PDO mapping axis 1: SS2_1 error
	eAX580x_ERROR_FAULT_PDO_MAPPING_SSR_1_K1		 	:= 16#072C,	// PDO mapping axis 1: SSR_1 error
	eAX580x_ERROR_FAULT_PDO_MAPPING_SDIp_K1				:= 16#072D,	// PDO mapping axis 1: SDIp error
	eAX580x_ERROR_FAULT_PDO_MAPPING_SDIn_K1				:= 16#072E,	// PDO mapping axis 1: SDIn error
	eAX580x_ERROR_FAULT_PDO_MAPPING_Error_ACK_K1	 	:= 16#072F,	// PDO mapping axis 1: Error_ACK error
	eAX580x_ERROR_FAULT_PDO_MAPPING_Error_CRC0			:= 16#0730,	// PDO mapping axis 1/2: FSOE CRC0 error
	eAX580x_ERROR_FAULT_PDO_MAPPING_STO_K2				:= 16#0731,	// PDO mapping axis 2: STO error 
	eAX580x_ERROR_FAULT_PDO_MAPPING_SS1_1_K2			:= 16#0732,	// PDO mapping axis 2: Error SS1_1 
	eAX580x_ERROR_FAULT_PDO_MAPPING_SS2_1_K2			:= 16#0733,	// PDO mapping axis 2: Error SS2_1 
	eAX580x_ERROR_FAULT_PDO_MAPPING_SOS_1_K2			:= 16#0734,	// PDO mapping axis 2: SS2_1 error
	eAX580x_ERROR_FAULT_PDO_MAPPING_SSR_1_K2			:= 16#0735,	// PDO mapping axis 2: SSR_1 error
	eAX580x_ERROR_FAULT_PDO_MAPPING_SDIp_K2				:= 16#0736,	// PDO mapping axis 2: SDIp error
	eAX580x_ERROR_FAULT_PDO_MAPPING_SDIn_K2				:= 16#0737,	// PDO mapping axis 2: SDIn error
	eAX580x_ERROR_FAULT_PDO_MAPPING_Error_ACK_K2	 	:= 16#0738,	// PDO mapping axis 2: Error_ACK error
	eAX580x_ERROR_FAULT_PDO_MAPPING_Error_CRC1			:= 16#0739,	// PDO mapping axis 2: FSOE CRC1 error
	eAX580x_ERROR_FAULT_PDO_MAPPING_Error_ConnID		:= 16#073A,	// PDO mapping axis 1/2: FSOE ConnID error
	eAX580x_ERROR_FAULT_PDO_MAPPING_SSM_1_K1			:= 16#073B,	// PDO mapping axis 1: SSM_1_K1 error
	eAX580x_ERROR_FAULT_PDO_MAPPING_SSM_1_K2			:= 16#073C,	// PDO mapping axis 2: SSM_1_K2 error
	eAX580x_ERROR_FAULT_PDO_MAPPING_SSM_2_K1			:= 16#073D,	// PDO mapping axis 1: SSM_2_K1 error
	eAX580x_ERROR_FAULT_PDO_MAPPING_SSM_2_K2			:= 16#073E,	// PDO mapping axis 2: SSM_2_K2 error
	eAX580x_ERROR_FAULT_WRONG_MOTORCONSTR_UCTIONTYPE_K1	:= 16#0740,	// Register communication: parameterized motor type for axis 1 does not correspond to the connected motor.
	eAX580x_ERROR_FAULT_UNKNOWN_MOTOR_TYPE_K1			:= 16#0741,	// Register communication: parameterized motor type for axis 1 is unknown
	eAX580x_ERROR_FAULT_WRONG_MOTORCONSTR_UCTIONTYPE_K2	:= 16#0742,	// Register communication: parameterized motor type for axis 2 does not correspond to the connected motor.
	eAX580x_ERROR_FAULT_UNKNOWN_MOTOR_TYPE_K2			:= 16#0743,	// Register communication: parameterized motor type for axis 2 is unknown.
	eAX580x_ERROR_FAULT_NUM_OF_POLEPAIRS_K1				:= 16#0744,	// Register communication: parameterized number of pole pairs for axis 1 does not correspond to the connected motor.
	eAX580x_ERROR_FAULT_NUM_OF_POLEPAIRS_K2				:= 16#0745,	// Register communication: parameterized number of pole pairs for axis 2 does not correspond to the connected motor.
	eAX580x_ERROR_FAULT_WRONG_MOTOR_CONFIGURED_K1		:= 16#0746,	// Register communication: parameterized motor type for axis 1 does not correspond to the connected motor.
	eAX580x_ERROR_FAULT_WRONG_MOTOR_CONFIGURED_K2		:= 16#0747,	// Register communication: parameterized motor type for axis 2 does not correspond to the connected motor
	eAX580x_ERROR_FAULT_RXPDO_LENGTH					:= 16#0748,	// PDO mapping: RXPDO length is wrong.
	eAX580x_ERROR_FAULT_TXPDO_LENGTH					:= 16#0749,	// PDO mapping: TXPDO length is wrong.
	eAX580x_ERROR_FAULT_UNKNOWN_RXPDO_INDEX				:= 16#074A,	// PDO mapping: RXPDO index is unknown 
	eAX580x_ERROR_FAULT_UNKNOWN_TXPDO_INDEX				:= 16#074B,	// PDO mapping: TXPDO index is unknown 
	eAX580x_ERROR_FAULT_WRONG_NUMBER_OF_AXLE			:= 16#074C,	// The parameterized number of axes does not correspond to the number detected.
	eAX580x_ERROR_FAULT_CRC_INIT_C1						:= 16#1001,	// An incorrect checksum at µC1 was determined during PowerOn reset.
	eAX580x_ERROR_FAULT_CRC_INIT_C2						:= 16#1002,	// An incorrect checksum at µC2 was determined during PowerOn reset.
	eAX580x_ERROR_FAULT_CRC_C1							:= 16#1003,	// An incorrect checksum was determined for µC1 during operation.
	eAX580x_ERROR_FAULT_CRC_C2							:= 16#1004,	// An incorrect checksum was determined for µC2 during operation.
	eAX580x_ERROR_FAULT_RAM_C1							:= 16#1011,	// An error occurred during the RAM test of µC1.
	eAX580x_ERROR_FAULT_RAM_C2							:= 16#1012,	// An error occurred during the RAM test of µC2.
	eAX580x_ERROR_FAULT_RAM_CHECKERBOARD_C1				:= 16#1013,	// An error occurred during the RAM test of µC1.
	eAX580x_ERROR_FAULT_RAM_CHECKERBOARD_C2				:= 16#1014,	// An error occurred during the RAM test of µC2.
	eAX580x_ERROR_FAULT_GLBL_TMR						:= 16#1021,	// The global timer is not working correctly.
	eAX580x_ERROR_FAULT_SPLIM1							:= 16#1031,	// Stack overruns are no longer being intercepted correctly.
	eAX580x_ERROR_FAULT_SPLIM2 							:= 16#1032,	// Stack overruns are no longer being intercepted correctly.
	eAX580x_ERROR_FAULT_OPCT_GRP_C1						:= 16#1100,	// The opcode test for µC1 has failed.
	eAX580x_ERROR_FAULT_OPCT_GRP_C2						:= 16#1300,	// The opcode test for µC2 has failed.
	eAX580x_ERROR_FAULT_ESS_CRC_C1						:= 16#1801,	// Different check sums were determined in the TwinSAFE telegrams.
	eAX580x_ERROR_FAULT_ESS_CRC_C2						:= 16#1802,	// Different check sums were determined in the TwinSAFE telegrams.
	eAX580x_ERROR_FAULT_SW_MAIN1_C1						:= 16#1803,	// The default case of the main loop of µC1 was called.
	eAX580x_ERROR_FAULT_SW_MAIN1_C2						:= 16#1804,	// The default case of the main loop of µC2 was called.
	eAX580x_ERROR_FAULT_ESLCONID_PRJCRCRD				:= 16#1805,	// The Connection ID is not zero when reading the project CRC.
	eAX580x_ERROR_FAULT_ESLCONID_PRJCRCWR				:= 16#1806,	// The Connection ID is not zero when writing the project CRC.
	eAX580x_ERROR_FAULT_SIZE_EEVONDOR_EXID 				:= 16#1807,	// An address was accessed that lies outside the vendor range in the EEPROM. 
	eAX580x_ERROR_FAULT_COM_C1C2						:= 16#5100,	// Communication between µC1 and µC2 is disturbed.
	eAX580x_ERROR_FAULT_ISR_SNT_FEEDBACK				:= 16#5101,	// High priority ISR: communication interrupted: switched mode power supply feedback 
	eAX580x_ERROR_FAULT_ISR_ANGLE_K1					:= 16#5102,	// High priority ISR: communication interrupted: axis 1 angle 
	eAX580x_ERROR_FAULT_ISR_ANGLE_K2					:= 16#5103,	// High priority ISR: communication interrupted: axis 2 angle 
	eAX580x_ERROR_FAULT_ISR_DELTA_K1					:= 16#5104,	// High priority ISR: communication interrupted: axis 1 distance travelled 
	eAX580x_ERROR_FAULT_ISR_DELTA_K2					:= 16#5105,	// High priority ISR: communication interrupted: axis 2 distance travelled 
	eAX580x_ERROR_FAULT_ISR_VELO_K1						:= 16#5106,	// High priority ISR: communication interrupted: axis 1 velocity
	eAX580x_ERROR_FAULT_ISR_VELO_K2						:= 16#5107,	// High priority ISR: communication interrupted: axis 2 velocity
	eAX580x_ERROR_FAULT_ISR_TEST_FEEDBACK				:= 16#5108,	// High priority ISR: communication interrupted: feedback from switch-off channels
	eAX580x_ERROR_FAULT_TIMEOUT_REG_AX5000_CONTROL		:= 16#5109,	// Register communication: AX5000 does not answer in time: Controlword
	eAX580x_ERROR_FAULT_TIMEOUT_REG_AX5000_STATUS		:= 16#510A,	// Register communication: AX5000 does not answer in time: Statusword
	eAX580x_ERROR_FAULT_TIMEOUT_REG_AX5000_REGADR		:= 16#510B,	// Register communication: AX5000 does not answer in time: Register address
	eAX580x_ERROR_FAULT_TIMEOUT_REG_AX5000_REGDATA		:= 16#510C,	// Register communication: AX5000 does not answer in time: Register data
	eAX580x_ERROR_FAULT_TIMEOUT_REG_AX5000_CRC			:= 16#510D,	// Register communication: AX5000 does not answer in time: CRC
	eAX580x_ERROR_FAULT_UNKNOWN_AX5000_INTERFACE 		:= 16#510E,	// Register communication: unknown interface to the AX5000
	eAX580x_ERROR_FAULT_COMERROR_AX5000_INTERFACE		:= 16#510F,	// Register communication: the interface to the AX5000 has a communication error 
	eAX580x_ERROR_FAULT_WRITE_HW_VERSION_AX5805			:= 16#5110,	// Values could not be written to the register in the AX5000
	eAX580x_ERROR_FAULT_EXT_ADC_ADDRESS					:= 16#5114,	// High priority ISR: External ADC: an impermissible address was read
	eAX580x_ERROR_FAULT_REGISTER_AX5000_CRC_ERROR		:= 16#5115,	// Register communication with the AX5000: telegram has a CRC error.
	eAX580x_ERROR_FAULT_CYCLIC_AX5000_CRC_ERROR			:= 16#5116,	// High priority ISR: cyclic communication with the AX5000: telegram has a CRC error.
	eAX580x_ERROR_FAULT_UNKNOWN_REGISTER_ADDRESS	 	:= 16#5117,	// Register communication: Addressed register is unknown.
	eAX580x_ERROR_FAULT_AX5000_NOT_READY				:= 16#5118,	// High priority ISR: cyclic communication with the AX5000: AX5000 signals a communication error.
	eAX580x_ERROR_FAULT_C1C2_SYNC_LOST					:= 16#5119,	// High priority ISR: cyclic communication between µC1 and µC2: Communication error
	eAX580x_ERROR_FAULT_SET_MAPPED_STATE				:= 16#5C00,	// Mapped safety functions: error while setting the state.
	eAX580x_ERROR_FAULT_RESET_MAPPED_STATE				:= 16#5C01,	// Mapped safety functions: error while resetting the state.
	eAX580x_ERROR_FAULT_MAPPED_FUNCTION					:= 16#5C02,	// Mapped safety functions: invalid mapping, function does not exist.
	eAX580x_ERROR_FAULT_MAPPED_INSTANCE					:= 16#5C03,	// Mapped safety functions: invalid mapping, instance does not exist.
	eAX580x_ERROR_FAULT_STO_MODE						:= 16#5E02,	// The requested STO mode is invalid.
	eAX580x_ERROR_FAULT_UNDEFINED_ERRORREACTION			:= 16#5E04,	// Error reaction: invalid error reaction, error reaction does not exist.
	eAX580x_ERROR_FAULT_SDI_MODE						:= 16#5E03,	// The requested SDI mode is invalid.
	eAX580x_ERROR_FAULT_CRC_COMPARE_C1					:= 16#5F00,	// Incorrect checksum detected during comparison by µC1.
	eAX580x_ERROR_FAULT_CRC_COMPARE_C2					:= 16#5F01,	// Incorrect checksum detected during comparison by µC2.
	eAX580x_ERROR_FAULT_TMR2_INTERRUPT_C1				:= 16#5F02,	// MC_Test: Timer2 has triggered an interrupt on µC1. HighPrioISR was not called in time.
	eAX580x_ERROR_FAULT_TMR2_INTERRUPT_C2				:= 16#5F03,	// MC_Test: Timer2 has triggered an interrupt on µC2. HighPrioISR was not called in time.
	eAX580x_ERROR_FAULT_SWITCHOFF_TEST					:= 16#5F04,	// MC_Test: the test of the switch-off channels has failed.
	eAX580x_ERROR_FAULT_NO_SYNC 	 					:= 16#5F05,	// No SYNC signal 
	eAX580x_ERROR_FAULT_UNKNOWN_AXLE					:= 16#5F06,	// The requested axis is unknown.
	eAX580x_ERROR_FAULT_FPGA_C2							:= 16#5F07,	// The status of the FPGA is incorrect.
	eAX580x_ERROR_FAULT_ANGLE_FORMAT_C1					:= 16#5F08,	// The angles of µC1 read-in have the wrong format.
	eAX580x_ERROR_FAULT_ANGLE_FORMAT_C2					:= 16#5F09,	// The angles of µC2 read-in have the wrong format.
	eAX580x_ERROR_FAULT_SAFE_MAIN_STATE					:= 16#5F0A,	// Unknown state requested
	eAX580x_ERROR_FAULT_STARTUP_FAILED					:= 16#5F0B,	// Error during start-up.
	eAX580x_ERROR_FAULT_MOTION_DETECTION				:= 16#5F0C,	// Motion detection error
	eAX580x_ERROR_FAULT_PARAMETER_FSOE_VENDOR_ID	 	:= 16#6000,	// Incorrect vendor ID transmitted
	eAX580x_ERROR_FAULT_PARAMETER_FSOE_MODULE_IDENT		:= 16#6001,	// Incorrect module ID transmitted
	eAX580x_ERROR_FAULT_PARAMETER_FSOE_CRC	 			:= 16#6002	// CRC of the AX5805 parameters does not match the transmitted CRC (please check parameters, if necessary, activate System Manager configuration and reload safety project into the EL69xx).
);
END_TYPE

// ---- DUTs/HW/ST_AX580x_DiagnosticData.TcDUT
TYPE ST_AX580x_DiagnosticData EXTENDS ST_ELxxxx_Data:
STRUCT
	// Reason for switching off	
	CoE_0xFA82_01				: DWORD;
	CoE_0xFA82_02				: DWORD;
	CoE_0xFA82_03				: DWORD;
	CoE_0xFA82_04				: DWORD;
	// General diagnostic words
	// index 2->8 depend on contents of index 01 
	CoE_0xFA10_01				: DWORD;
	CoE_0xFA10_02				: DWORD;
	CoE_0xFA10_03				: DWORD;
	CoE_0xFA10_04				: DWORD;
	CoE_0xFA10_05				: DWORD;
	CoE_0xFA10_06				: DWORD;	
	// Reason for shut-down if index 01 == 0
	// Axis 1
	bAxis1_NoErrorReaction		: BOOL;
	bAxis1_STOErrorReaction		: BOOL;
	bAxis1_SS1ErrorReaction		: BOOL;
	CoE_0xFA10_07				: DWORD;
	// Axis 2
	bAxis2_NoErrorReaction		: BOOL;
	bAxis2_STOErrorReaction		: BOOL;
	bAxis2_SS1ErrorReaction		: BOOL;
	CoE_0xFA10_08				: DWORD;	
	// Other error on FA10_xx
	bError_FA10_xx				: BOOL;
END_STRUCT
END_TYPE

// ---- DUTs/HW/ST_EL1904_DiagnosticData.TcDUT
TYPE ST_EL1904_DiagnosticData EXTENDS ST_ELxxxx_Data:
STRUCT
	bInput1				: BOOL;
	bInput2				: BOOL;
	bInput3				: BOOL;
	bInput4				: BOOL;
	(* 800E:0A Sensor test error - Error during the sensor test *)
	bSensorTestError1	: BOOL; (* Error at input 1 *)
	bSensorTestError2	: BOOL; (* Error at input 2 *)
	bSensorTestError3	: BOOL; (* Error at input 3 *)
	bSensorTestError4	: BOOL; (* Error at input 4 *)
	(* 800E:0B Error during two-channel evaluation - Error during the contiguous evaluation of two channels, 
													i.e. the two channels contradict each other. *)
	b2ChEvError1		: BOOL; (* Error in the first input pair *)
	b2ChEvError2		: BOOL; (* Error in the second input pair *)
	(* 800E:0C Error in the safety mat operation mode: input pair disagree - Error in the input pair *)
	b2ChMatError1		: BOOL; (* Error in the first input pair  - BIT 0, 1 - 11 bin *)
	b2ChMatError2		: BOOL; (* Error in the second input pair - BIT 2, 3 - 11 bin *)
	(* 800E:0D Error in the safety mat operation mode: external supply - Error in the test pulses in the safety mat operating mode; 
																		i.e. the terminal has detected an external supply. *)
	bTestPulsesError1	: BOOL; (* Error at input 1 *)
	bTestPulsesError2	: BOOL; (* Error at input 2 *)
	bTestPulsesError3	: BOOL; (* Error at input 3 *)
	bTestPulsesError4	: BOOL; (* Error at input 4 *)
END_STRUCT
END_TYPE

// ---- DUTs/HW/ST_EL2904_DiagnosticData.TcDUT
TYPE ST_EL2904_DiagnosticData EXTENDS ST_ELxxxx_Data:
STRUCT
	(* FA80:03 Temperature Outputs - Temperature measurement (right board)*)
	wTemperatureOut		: WORD;
	bOutput1			: BOOL; (* Output 1 *)
	bOutput2			: BOOL; (* Output 2 *)
	bOutput3			: BOOL; (* Output 3 *)
	bOutput4			: BOOL; (* Output 4 *)
	(* 800E:0C Error at the output *)
	(* External supply or cross-circuit.  These diagnostic messages are displayed only if Current Measurement active = false. *)
	bOutputCross1		: BOOL; (* Output 1 *)
	bOutputCross2		: BOOL; (* Output 2 *)
	bOutputCross3		: BOOL; (* Output 3 *)
	bOutputCross4		: BOOL; (* Output 4 *)
	(* Open load or current below minimum value of 20 mA or current above maximum value of 500 mA *)
	bOutputOpen1		: BOOL; (* Output 1 *)
	bOutputOpen2		: BOOL; (* Output 2 *)
	bOutputOpen3		: BOOL; (* Output 3 *)
	bOutputOpen4		: BOOL; (* Output 4 *)
	(*800E:0D Supply error*)
	bFieldVoltH			: BOOL; (* Field voltage too high *)
	bFieldVoltL			: BOOL; (* Field voltage too low *)
	(*800E:0E Temperature error*)
	bTHUC1				: BOOL; (* Overtemperature uC1 *)
	bTHUC2				: BOOL; (* Overtemperature uC2 *)
	bTOutBoardH			: BOOL; (* Overtemperature of the output board *)
	bTLUC1				: BOOL; (* Temperature too low uC1 *)
	bTLUC2				: BOOL; (* Temperature too low uC2 *)
	bTOutBoardL			: BOOL; (* Temperature of the output board too low *)
	bTDiffProcBoard		: BOOL; (* Temperature difference on the processor board too large *)
	bTDiffBoards		: BOOL; (* Temperature difference between the boards is too large *)
END_STRUCT
END_TYPE

// ---- DUTs/HW/ST_EL6900_DiagnosticData.TcDUT
TYPE ST_EL6900_DiagnosticData EXTENDS ST_ELxxxx_Data:
STRUCT
	wSafetyProjectState		: WORD; 	(* F100:01 *)
	eSAFETY_ProjectState	: E_SAFETY_ProjectState;
	dwProjectCRC			: DWORD;	(* F980:03 *)
	sProjectCRC				: STRING(4);
	wVccPrimaryMC			: WORD;		(* FA80:03 *)
	wVccSecondaryMC			: WORD;		(* FA80:04 *)
	(* FA00:03 *)
	(* Temperature error: 	16#0005 - Maximum temperature exceeded 
							16#0006 - Temperature fell below minimum 
							16#0007 - Temperature difference between the measuring points exceeded
		Supply error		16#0101 - max. supply voltage uC1 exceeded
							16#0102 - max. supply voltage uC2 exceeded
							16#0103 - voltage fell below min. supply voltage uC1 
							16#0104 - voltage fell below min. supply voltage uC2 *)
	bTempMax				: BOOL;
	bTempMin				: BOOL;
	bTempDiff				: BOOL;
	bSuppVoltuMaxC1			: BOOL;
	bSuppVoltuMaxC2			: BOOL;
	bSuppVoltuMinC1			: BOOL;
	bSuppVoltuMinC2			: BOOL;
END_STRUCT
END_TYPE

// ---- DUTs/HW/ST_EL6900_StatusData.TcDUT
TYPE ST_EL6900_StatusData :
STRUCT
	dwStatusConnections			: DWORD; 										(* 2110:0 *) (* Liczba polaczen *)
	arrstStatusConnections		: ARRAY [1..128] OF ST_SAFETYStatusConnection; 	(* 2110:01-80 *)
	dwStatusGroups				: DWORD; 										(* 2120:0 *) (* Liczba grup *)
	arrstStatusGroups			: ARRAY [1..32] OF ST_SAFETYStatusGroup; 		(* 2120:01-20 *)
	dwStatusFunctionBlocks		: DWORD; 										(* 2130:0 *) (* Liczba blokow *)
	arrstStatusFunctionBlocks	: ARRAY [1..255] OF ST_SAFETY_FBStatus; 		(* 2130:01-FF *)
END_STRUCT
END_TYPE

// ---- DUTs/HW/ST_ELxxxx_Data.TcDUT
TYPE ST_ELxxxx_Data :
STRUCT
	sDeviceName				: STRING;	(* 1008 *)
	sHardwareVersion		: STRING;	(* 1009 *)
	sSoftwareVersion		: STRING;	(* 100A *)
	dwFSoEAddress			: DWORD;	(* F980:01 *)
	dwSerialNumber			: DWORD;	(* F980:02 *)
	sSerialNumber			: STRING(8);	
	wTemperaturePrimaryMC	: WORD;		(* FA80:01 Temperature 1 - Temperature measurement 1 *)
	wTemperatureSecondaryMC	: WORD;		(* FA80:02 Temperature 2 - Temperature measurement 2 *)
	bGeneralError			: BOOL; 	(* Gdy wystapi chociaz jeden Error *)
END_STRUCT
END_TYPE

// ---- DUTs/Others/E_SAFETY_ConnectionDiag.TcDUT
TYPE E_SAFETY_ConnectionDiag :
(* Only 4 least significant bits of diagnostic information for a connection. *)
(	eSAFETY_ConnectDiag_WithoutErrors			:=	2#0000,
	eSAFETY_ConnectDiag_InvalidCommmand			:=	2#0001,
	eSAFETY_ConnectDiag_UnknownCommand			:=	2#0010,
	eSAFETY_ConnectDiag_InvalidConnectionID		:=	2#0011,
	eSAFETY_ConnectDiag_InvalidCRC				:=	2#0100,
	eSAFETY_ConnectDiag_WatchdogTimeElapsed		:=	2#0101,
	eSAFETY_ConnectDiag_InvalidFSoEAddress		:=	2#0110,
	eSAFETY_ConnectDiag_InvalidData				:=	2#0111,
	eSAFETY_ConnectDiag_InvalidCommParamLength	:=	2#1000,
	eSAFETY_ConnectDiag_InvalidCommParams		:=	2#1001,
	eSAFETY_ConnectDiag_InvalidUserParamLength	:=	2#1010,
	eSAFETY_ConnectDiag_InvalidUserParams		:=	2#1011,
	eSAFETY_ConnectDiag_FSoEMasterReset			:=	2#1100,
	eSAFETY_ConnectDiag_ModuleError				:=	2#1101,
	eSAFETY_ConnectDiag_EL290xError				:=	2#1110,
	eSAFETY_ConnectDiag_SlaveNotYetStarted		:=	2#1111
);
END_TYPE

// ---- DUTs/Others/E_SAFETY_ConnectionState.TcDUT
TYPE E_SAFETY_ConnectionState :
(
	eSAFETY_ConnectionState_Unknown		:= 0,
	eSAFETY_ConnectionState_Reset 		:= 100,
	eSAFETY_ConnectionState_Session 	:= 101,
	eSAFETY_ConnectionState_Connection	:= 102,
	eSAFETY_ConnectionState_Parameter	:= 103,
	eSAFETY_ConnectionState_Data		:= 104,
	eSAFETY_ConnectionState_Shutdown	:= 105
);
END_TYPE

// ---- DUTs/Others/E_SAFETY_GroupState.TcDUT
TYPE E_SAFETY_GroupState :
(
	eSAFETY_GroupState_UNKNOWN		:= 0,
	eSAFETY_GroupState_RUN 			:= 1,
	eSAFETY_GroupState_STOP 		:= 2,
	eSAFETY_GroupState_SAFE			:= 3,
	eSAFETY_GroupState_ERROR		:= 4,
	eSAFETY_GroupState_RESET		:= 5
);
END_TYPE

// ---- DUTs/Others/E_SAFETY_ProjectState.TcDUT
TYPE E_SAFETY_ProjectState :
(
	eSAFETY_ProjectState_OFFLINE 	:= 0,
	eSAFETY_ProjectState_RUN		:= 1,
	eSAFETY_ProjectState_STOP 		:= 2,
	eSAFETY_ProjectState_START 		:= 3,
	eSAFETY_ProjectState_RESTORE	:= 4,
	eSAFETY_ProjectState_FAULT 		:= 5
);
END_TYPE

// ---- DUTs/Others/ST_SAFETYGroupIO.TcDUT
TYPE ST_SAFETYGroupIO :
STRUCT
	RUN_STOP 				AT %Q* : BIT := TRUE;
	ERR_Ack 				AT %Q* : BIT;
	FB_ERR 					AT %I* : BIT;
	COM_ERR 				AT %I* : BIT;
	OUT_ERR 				AT %I* : BIT; (* Only in KL6904  *)
END_STRUCT
END_TYPE

// ---- DUTs/Others/ST_SAFETYStatusConnection.TcDUT
TYPE ST_SAFETYStatusConnection :
STRUCT
	dwStatusConnection			: DWORD;
	BState						: BYTE;
	BDiagnosis					: BYTE;	(*	xxxx 0001  Invalid command 
											xxxx 0010  Unknown command 
											xxxx 0011  Invalid connection ID 
											xxxx 0100  Invalid CRC 
											xxxx 0101  Watchdog time elapsed 
											xxxx 0110  Invalid FSoE address 
											xxxx 0111  Invalid data 
											xxxx 1000  Invalid communication parameter length 
											xxxx 1001  Invalid communication parameters 
											xxxx 1010  Invalid user parameter length 
											xxxx 1011  Invalid user parameters 
											xxxx 1100  FSoE master reset 
											xxxx 1101  Module error detected on slave, with option "Module error is ComError" activated 
											xxxx 1110  Module error detected on EL290x, with option "Error acknowledge active" activated 
											xxxx 1111  Slave not yet started, or unexpected error argument 
											xxx1 xxxx  FSoE slave error detected 
											xx1x xxxx  FSoE slave reports Failsafe Value active 
											x1xx xxxx  StartUp 
											1xxx xxxx  FSoE master reports Failsafe Value active *)
	eSAFETY_ConnectionDiag0F	: E_SAFETY_ConnectionDiag;
	sSAFETY_ConnectionDiagF0	: STRING(4);
	BSAFETY_ConnectionDiagF0	: BYTE;
	eSAFETY_ConnectionState		: E_SAFETY_ConnectionState;
END_STRUCT
END_TYPE

// ---- DUTs/Others/ST_SAFETYStatusGroup.TcDUT
TYPE ST_SAFETYStatusGroup :
STRUCT
	dwStatusGroup					: DWORD;
	BState							: BYTE;
	BDiagnosis						: BYTE;
	BInputs							: BYTE;
	BOutputs						: BYTE;
	eSAFETY_GroupState				: E_SAFETY_GroupState;
	bRUN_STOP 						: BOOL;
	bERR_Ack 						: BOOL;
	bFB_ERR 						: BOOL;
	bCOM_ERR 						: BOOL;
	bOUT_ERR 						: BOOL;
END_STRUCT
END_TYPE

// ---- Version/Global_Version.TcGVL
{attribute 'TcGenerated'}
// This function has been automatically generated from the project information.
VAR_GLOBAL CONSTANT
	{attribute 'const_non_replaced'}
	{attribute 'linkalways'}
	stLibVersion_TC3SafetyDiag : ST_LibVersion := (iMajor := 2, iMinor := 7, iBuild := 0, iRevision := 0, sVersion := '2.7.0');
END_VAR

// ---- POUs/Others/I_ErrorHandling.TcIO
INTERFACE I_ErrorHandling

PROPERTY P_Error : bool
GET
END_GET
END_PROPERTY

PROPERTY P_ErrorID : udint
GET
END_GET
END_PROPERTY

METHOD ToString : String(255)
VAR_INPUT
END_VAR
END_METHOD

END_INTERFACE

// ---- POUs/MAINSafety.TcPOU
PROGRAM MAINSafety
VAR CONSTANT
	sNetID: T_AmsNetId := '10.24.33.33.2.1'; // EtherCAT Master AMS NetID
END_VAR
VAR
	(* I/O *)
	bEnable 			AT %I*	: BOOL; (* Pozwolenie na prace z SAFETY ESTOP *)
	stSAFETYGroupIO				: ST_SAFETYGroupIO;
	fbSAFETY_AutoGroupErrACK	: FB_SAFETY_AutoGroupErrACK;
	(* HW diagnostic *)
	fbEL1904_DiagnosticData		: FB_EL1904_DiagnosticData;
	stEL1904_DiagnosticData		: ST_EL1904_DiagnosticData;
	fbEL2904_DiagnosticData		: FB_EL2904_DiagnosticData;
	stEL2904_DiagnosticData		: ST_EL2904_DiagnosticData;
	fbEL6900_DiagnosticData		: FB_EL6900_DiagnosticData;
	stEL6900_DiagnosticData		: ST_EL6900_DiagnosticData;
	(* SAFETY project diagnostic *)
	fbEL6900_StatusData			: FB_EL6900_StatusData;
	stEL6900_StatusData			: ST_EL6900_StatusData;
	(* FBs conversion *)
	stSAFETY_FBESTOP			: ST_SAFETY_FBESTOP;
	stSAFETY_FBTwoHand			: ST_SAFETY_FBTWOHAND;
	stSAFETY_FBRS				: ST_SAFETY_FBRS;
	stSAFETY_FBTOF				: ST_SAFETY_FBTOF;
	stSAFETY_FBOPMODE			: ST_SAFETY_FBOPMODE;
	stSAFETY_FBMUTING			: ST_SAFETY_FBMUTING;
	stSAFETY_FBMON				: ST_SAFETY_FBMON;
	stSAFETY_FBDECOUPLE			: ST_SAFETY_FBDECOUPLE;
	stSAFETY_FBAND				: ST_SAFETY_FBAND;
	stSAFETY_FBOR				: ST_SAFETY_FBOR;
	(* Other *)
	tonDelay					: TON;
	rtInit						: R_TRIG;
	ftEL1904DiagEnd				: F_TRIG;
	ftEL2904DiagEnd				: F_TRIG;
	ftEL6900DiagEnd				: F_TRIG;
	ftEL6900StatusEnd			: F_TRIG;
END_VAR

tonDelay(IN := TRUE, PT := T#10s); // TON
rtInit(CLK := tonDelay.Q); // R_TRIG
fbSAFETY_AutoGroupErrACK(stSAFETYGroupIO := stSAFETYGroupIO); // FB_SAFETY_AutoGroupErrACK
fbEL1904_DiagnosticData(sNetId := sNetID, uiSlaveAddr := 1006, bExecute := rtInit.Q OR ftEL6900StatusEnd.Q); // FB_EL1904_DiagnosticData
stEL1904_DiagnosticData := fbEL1904_DiagnosticData.stEL1904_DiagnosticData;
ftEL1904DiagEnd(CLK := fbEL1904_DiagnosticData.bBusy); // F_TRIG
fbEL2904_DiagnosticData(sNetId := sNetID, uiSlaveAddr := 1007, bExecute := ftEL1904DiagEnd.Q); // FB_EL2904_DiagnosticData
stEL2904_DiagnosticData := fbEL2904_DiagnosticData.stEL2904_DiagnosticData;
ftEL2904DiagEnd(CLK := fbEL2904_DiagnosticData.bBusy); // F_TRIG
fbEL6900_DiagnosticData(sNetId := sNetID, uiSlaveAddr := 1005, bExecute := ftEL2904DiagEnd.Q); // FB_EL6900_DiagnosticData
stEL6900_DiagnosticData := fbEL6900_DiagnosticData.stEL6900_DiagnosticData;
ftEL6900DiagEnd(CLK := fbEL6900_DiagnosticData.bBusy); // F_TRIG
fbEL6900_StatusData(
    sNetId := sNetID,
    uiSlaveAddr := fbEL6900_DiagnosticData.uiSlaveAddr,
    bExecute := ftEL6900DiagEnd.Q); // FB_EL6900_StatusData
stEL6900_StatusData := fbEL6900_StatusData.stEL6900_StatusData;
ftEL6900StatusEnd(CLK := fbEL6900_StatusData.bBusy); // F_TRIG

END_PROGRAM

// ---- POUs/Others/FB_SAFETY_AutoGroupErrACK.TcPOU
FUNCTION_BLOCK FB_SAFETY_AutoGroupErrACK
VAR_IN_OUT
	stSAFETYGroupIO: ST_SAFETYGroupIO;
END_VAR

stSAFETYGroupIO.ERR_Ack := stSAFETYGroupIO.FB_ERR OR stSAFETYGroupIO.COM_ERR OR stSAFETYGroupIO.OUT_ERR;

END_FUNCTION_BLOCK

// ---- POUs/HW/FB_EL1904_DiagnosticData.TcPOU
(****************************************************************************************)
(*							Beckhoff Automation Poland									*)
(*									30.01.2017											*)
(*			Blok funkcyjny pobierający informacje diagnostyczne z modułu EL1904			*)
(*			v2.5:																		*)
(*				- bReset, wErrorCount, ACT_Reset zmiana nazw pozostalych akcji			*)
(*				- usunieta zmienna sPath												*)
(*			v2.4:																		*)
(*				- obsluga bledu															*)
(*			v2.3:																		*)
(*				- dostosowano do rozbudowanej struktury									*)
(*			v1.2:																		*)
(*				- uruchamianie zboczem narastającym bExecute							*)	
(*______________________________________________________________________________________*)
FUNCTION_BLOCK FB_EL1904_DiagnosticData IMPLEMENTS I_ErrorHandling
VAR_INPUT
	sNetId						: T_AmsNetId;					(* Adres mastera EtherCAT *)
	uiSlaveAddr					: UINT;							(* Adres slave EtherCAT modułu EL1904 *)
	bExecute					: BOOL;							(* Zbocze narastające aktywuje komende *)
	bReset						: BOOL;							(* 	*)
END_VAR
VAR_OUTPUT
	stEL1904_DiagnosticData		: ST_EL1904_DiagnosticData;		(* Wyjściowa struktura danych *)
	bBusy						: BOOL;							(* Wyjście jest ustawione gdy aktualnie wykonywana jest komenda *)
	bError						: BOOL;							(* Wyjście jest ustawione gdy wystąpił błąd *) 
	udiErrorId					: UDINT;						(* Kod błedu *)
	bNewData					: BOOL;							(* Po otrzymaniu nowych danych przyjmuje wartość TRUE na jeden cykl *)
END_VAR
VAR
	fbEcCoESdoRead				: FB_EcCoESdoRead;
	stTempData					: ST_EL1904_DiagnosticData;		(* Tymczasowa struktura danych *)
	BSubIndex					: BYTE;
	wIndex						: WORD;
	iStep						: INT;
	pDstBuf						: PVOID;
	cbBufLen					: UDINT;
	rtExecute					: R_TRIG;
	rtError						: R_TRIG;
	rtReset						: R_TRIG;
	bRead						: BOOL;							(* Odczyt *)
	wTemp_800E_0A				: WORD;							(* Wartosc tymczasowa *)
	wTemp_800E_0B				: WORD;							(* Wartosc tymczasowa *)
	wTemp_800E_0C				: WORD;							(* Wartosc tymczasowa *)
	wTemp_800E_0D				: WORD;							(* Wartosc tymczasowa *)
	wErrorCount					: WORD;							// Licznik bledow
END_VAR

ACT_Reset(); 									// Wywolanie akcji resetu

rtExecute(CLK:=bExecute);

CASE iStep OF	
	(* Wspolne *)	
	0:
												(* Odczyt nazwy modułu *)
		bNewData	:= FALSE;
		bRead		:= FALSE;
		IF rtExecute.Q THEN
			bBusy			:= TRUE;
			bError			:= FALSE;
			udiErrorId		:= 0;
			wIndex 			:= 16#1008;
			BSubIndex 		:= 0;
			pDstBuf 		:= ADR (stTempData.sDeviceName);
			cbBufLen 		:= SIZEOF(stTempData.sDeviceName);
			bRead			:= TRUE;
			iStep			:= iStep + 10;
		END_IF
	10:												(* Odczyt wersji HW *)
		bRead		:= FALSE;
		IF NOT fbEcCoESdoRead.bBusy AND NOT fbEcCoESdoRead.bError THEN
			wIndex 			:= 16#1009;
			BSubIndex 		:= 0;
			pDstBuf 		:= ADR (stTempData.sHardwareVersion);
			cbBufLen 		:= SIZEOF(stTempData.sHardwareVersion);
			bRead			:= TRUE;
			iStep			:= iStep + 10;
		END_IF
	20:												(* Odczyt wersji SW *)
		bRead				:= FALSE;
		IF NOT fbEcCoESdoRead.bBusy AND NOT fbEcCoESdoRead.bError THEN
			wIndex 			:= 16#100A;
			BSubIndex 		:= 0;
			pDstBuf 		:= ADR (stTempData.sSoftwareVersion);
			cbBufLen 		:= SIZEOF(stTempData.sSoftwareVersion);
			bRead			:= TRUE;
			iStep			:= iStep + 10;
		END_IF
	30:												(* Odczyt adresu FSoE *)
		bRead				:= FALSE;
		IF NOT fbEcCoESdoRead.bBusy AND NOT fbEcCoESdoRead.bError THEN
			wIndex 			:= 16#F980;
			BSubIndex 		:= 1;
			pDstBuf 		:= ADR (stTempData.dwFSoEAddress);
			cbBufLen 		:= SIZEOF(stTempData.dwFSoEAddress);
			bRead			:= TRUE;
			iStep			:= iStep + 10;
		END_IF;
	40:												(* Odczyt numeru seryjnego *)
		bRead				:= FALSE;
		IF NOT fbEcCoESdoRead.bBusy AND NOT fbEcCoESdoRead.bError THEN
			wIndex 			:= 16#F980;
			BSubIndex 		:= 2;
			pDstBuf 		:= ADR (stTempData.dwSerialNumber);
			cbBufLen 		:= SIZEOF(stTempData.dwSerialNumber);
			bRead			:= TRUE;
			iStep			:= iStep + 10;
		END_IF
	50:												(* Odczyt Temperature measurement 1 *)
		bRead				:= FALSE;
		IF NOT fbEcCoESdoRead.bBusy AND NOT fbEcCoESdoRead.bError THEN
			wIndex 			:= 16#FA80;
			BSubIndex 		:= 1;
			pDstBuf 		:= ADR (stTempData.wTemperaturePrimaryMC);
			cbBufLen 		:= SIZEOF(stTempData.wTemperaturePrimaryMC);
			bRead			:= TRUE;
			iStep			:= iStep + 10;
		END_IF
	60:												(* Odczyt Temperature measurement 2 *)
		bRead				:= FALSE;
		IF NOT fbEcCoESdoRead.bBusy AND NOT fbEcCoESdoRead.bError THEN
			wIndex 			:= 16#FA80;
			BSubIndex 		:= 2;
			pDstBuf 		:= ADR (stTempData.wTemperatureSecondaryMC);
			cbBufLen 		:= SIZEOF(stTempData.wTemperatureSecondaryMC);
			bRead			:= TRUE;
			iStep			:= iStep + 10;
		END_IF
	(*Charakterystyczne dla modulu *)
	70:												(* Odczyt DI 1 *)
		bRead				:= FALSE;
		IF NOT fbEcCoESdoRead.bBusy AND NOT fbEcCoESdoRead.bError THEN
			wIndex 			:= 16#6001;
			BSubIndex 		:= 1;
			pDstBuf 		:= ADR(stTempData.bInput1);
			cbBufLen 		:= SIZEOF(stTempData.bInput1);
			bRead			:= TRUE;
			iStep			:= iStep + 10;
		END_IF
	80:												(* Odczyt DI 2 *)
		bRead				:= FALSE;
		IF NOT fbEcCoESdoRead.bBusy AND NOT fbEcCoESdoRead.bError THEN
			wIndex 			:= 16#6001;
			BSubIndex 		:= 2;
			pDstBuf 		:= ADR (stTempData.bInput2);
			cbBufLen 		:= SIZEOF(stTempData.bInput2);
			bRead			:= TRUE;
			iStep			:= iStep + 10;
		END_IF
	90:												(* Odczyt DI 3 *)
		bRead				:= FALSE;
		IF NOT fbEcCoESdoRead.bBusy AND NOT fbEcCoESdoRead.bError THEN
			wIndex 			:= 16#6001;
			BSubIndex 		:= 3;
			pDstBuf 		:= ADR (stTempData.bInput3);
			cbBufLen 		:= SIZEOF(stTempData.bInput3);
			bRead			:= TRUE;
			iStep			:= iStep + 10;
		END_IF
	100:											(* Odczyt DI 4 *)
		bRead				:= FALSE;
		IF NOT fbEcCoESdoRead.bBusy AND NOT fbEcCoESdoRead.bError THEN
			wIndex 			:= 16#6001;
			BSubIndex 		:= 4;
			pDstBuf 		:= ADR (stTempData.bInput4);
			cbBufLen 		:= SIZEOF(stTempData.bInput4);
			bRead			:= TRUE;
			iStep			:= iStep + 10;
		END_IF
	110:											(* Odczyt 800E 0A *)
		bRead				:= FALSE;
		IF NOT fbEcCoESdoRead.bBusy AND NOT fbEcCoESdoRead.bError THEN
			wIndex 			:= 16#800E;
			BSubIndex 		:= 16#0A;
			pDstBuf 		:= ADR (wTemp_800E_0A);
			cbBufLen 		:= SIZEOF(wTemp_800E_0A);
			bRead			:= TRUE;
			iStep			:= iStep + 10;
		END_IF
	120:											(* Odczyt 800E 0B *)
		bRead				:= FALSE;
		IF NOT fbEcCoESdoRead.bBusy AND NOT fbEcCoESdoRead.bError THEN
			wIndex 			:= 16#800E;
			BSubIndex 		:= 16#0B;
			pDstBuf 		:= ADR (wTemp_800E_0B);
			cbBufLen 		:= SIZEOF(wTemp_800E_0B);
			bRead			:= TRUE;
			iStep			:= iStep + 10;
		END_IF
	130:											(* Odczyt 800E 0C *)
		bRead				:= FALSE;
		IF NOT fbEcCoESdoRead.bBusy AND NOT fbEcCoESdoRead.bError THEN
			wIndex 			:= 16#800E;
			BSubIndex 		:= 16#0C;
			pDstBuf 		:= ADR (wTemp_800E_0C);
			cbBufLen 		:= SIZEOF(wTemp_800E_0C);
			bRead			:= TRUE;
			iStep			:= iStep + 10;
		END_IF
	140:											(* Odczyt 800E 0D *)
		bRead				:= FALSE;
		IF NOT fbEcCoESdoRead.bBusy AND NOT fbEcCoESdoRead.bError THEN
			wIndex 			:= 16#800E;
			BSubIndex 		:= 16#0D;
			pDstBuf 		:= ADR (wTemp_800E_0D);
			cbBufLen 		:= SIZEOF(wTemp_800E_0D);
			bRead			:= TRUE;
			iStep			:= iStep + 10;
		END_IF
	150: (* Koniec odczytu *)
		bRead				:= FALSE;
		IF NOT fbEcCoESdoRead.bBusy AND NOT fbEcCoESdoRead.bError THEN
			iStep 			:= 200;
		END_IF
	
	200: (* Konwersje *)
		(* Zmiana numeru seryjnego na STRING *)
		stTempData.sSerialNumber 		:= '00000000';
		stTempData.sSerialNumber 		:= CONCAT(DELETE(stTempData.sSerialNumber, LEN(DWORD_TO_STRING(stTempData.dwSerialNumber)),1),DWORD_TO_STRING(stTempData.dwSerialNumber));
		stTempData.bSensorTestError1 	:= wTemp_800E_0A.0;
		stTempData.bSensorTestError2 	:= wTemp_800E_0A.1;
		stTempData.bSensorTestError3 	:= wTemp_800E_0A.2;
		stTempData.bSensorTestError4 	:= wTemp_800E_0A.3;
		(* Dekodowanie bitow w 800E *)
		stTempData.b2ChEvError1		 	:= wTemp_800E_0B.0;
		stTempData.b2ChEvError2	 		:= wTemp_800E_0B.1;
		stTempData.b2ChMatError1	 	:= wTemp_800E_0C.0 AND wTemp_800E_0C.1; (* Bit 1, 0 - 11bin - Error in the first input pair *)
		stTempData.b2ChMatError2	 	:= wTemp_800E_0C.2 AND wTemp_800E_0C.3; (* Bit 3, 2 - 11bin - Error in the second input pair *)
		stTempData.bTestPulsesError1 	:= wTemp_800E_0D.0;
		stTempData.bTestPulsesError2 	:= wTemp_800E_0D.1;
		stTempData.bTestPulsesError3 	:= wTemp_800E_0D.2;
		stTempData.bTestPulsesError4 	:= wTemp_800E_0D.3;
		(* General Error bit *)
		stTempData.bGeneralError := stTempData.bSensorTestError1 OR stTempData.bSensorTestError2 OR stTempData.bSensorTestError3 OR stTempData.bSensorTestError4 OR
									stTempData.b2ChEvError1 OR stTempData.b2ChEvError2 OR stTempData.b2ChMatError1 OR stTempData.b2ChMatError2 OR
									stTempData.bTestPulsesError1 OR stTempData.bTestPulsesError2 OR stTempData.bTestPulsesError3 OR stTempData.bTestPulsesError4;
		(* Przepisanie danych tymczasowych na wyjscie *)	
		stEL1904_DiagnosticData 		:= stTempData;
		(* Ustawienie flag i powrot do poczatku *)
		bBusy							:= FALSE;
		bNewData						:= TRUE;
		iStep 							:= 0;
	1000: (* ERROR *)
		wErrorCount 					:= wErrorCount + 1;			// Inkrementacja licznika bledow
		iStep 							:= 0;
END_CASE

fbEcCoESdoRead(
	sNetId		:= sNetId,
	nSlaveAddr	:= uiSlaveAddr,
	nSubIndex	:= BSubIndex,
	nIndex		:= wIndex,
	pDstBuf		:= pDstBuf,
	cbBufLen	:= cbBufLen,
	bExecute 	:= bRead);
	
ACT_Error();

ACTION ACT_Error:
rtError(CLK:= fbEcCoESdoRead.bError, Q=> );
IF rtError.Q THEN
	bBusy 			:= FALSE;
	bError 			:= TRUE;
	bRead			:= FALSE;
	udiErrorId 		:= fbEcCoESdoRead.nErrId;
	iStep 			:= 1000;
END_IF
END_ACTION

ACTION ACT_Reset:
rtReset(CLK:= bReset, Q=> );			// Wywolanie triggera, wykrycie zbocza narastajacego zmiennej wejsciowej bReset
IF rtReset.Q THEN
	bBusy						:= FALSE;
	bError						:= FALSE;
	bNewData					:= FALSE;
	bRead						:= FALSE;
	iStep						:= 0;
	udiErrorId					:= 0;
END_IF
END_ACTION

PROPERTY P_Error : BOOL
GET
END_GET
END_PROPERTY

PROPERTY P_ErrorID : UDINT
GET
END_GET
END_PROPERTY

{attribute 'object_name' := 'ToString'}
METHOD ToString : STRING(255)
END_METHOD

END_FUNCTION_BLOCK

